(* CoDeSys 2.3.9.42 project: komp_new2.pro *)
(* Libraries: Standard.lib 2.12.10 17:48:34, SYSLIBCALLBACK.LIB 2.12.10 17:48:32 *)

(* PLC configuration (modules and I/O channels)
0750-1405 16 DI 24V DC 3.0ms [Type_1_16_Channels] node 0, in %IB24 out %QB0 {INTTypePAAssignment = PLC; INTTypeModule = plugged}
  S4_1 AT %IX12.0 [BOOLOnX_I] Ch_1 Digital input
  S4_2 AT %IX12.1 [BOOLOnX_I] Ch_2 Digital input
  S5_1 AT %IX12.2 [BOOLOnX_I] Ch_3 Digital input
  S5_2 AT %IX12.3 [BOOLOnX_I] Ch_4 Digital input
  S6_1 AT %IX12.4 [BOOLOnX_I] Ch_5 Digital input
  S6_2 AT %IX12.5 [BOOLOnX_I] Ch_6 Digital input
  S7_1 AT %IX12.6 [BOOLOnX_I] Ch_7 Digital input
  S7_2 AT %IX12.7 [BOOLOnX_I] Ch_8 Digital input
  S8_1 AT %IX12.8 [BOOLOnX_I] Ch_9 Digital input
  S8_2 AT %IX12.9 [BOOLOnX_I] Ch_10 Digital input
  S9_1 AT %IX12.10 [BOOLOnX_I] Ch_11 Digital input
  S9_2 AT %IX12.11 [BOOLOnX_I] Ch_12 Digital input
  S10_1 AT %IX12.12 [BOOLOnX_I] Ch_13 Digital input
  S10_2 AT %IX12.13 [BOOLOnX_I] Ch_14 Digital input
  S11_1 AT %IX12.14 [BOOLOnX_I] Ch_15 Digital input
  S11_2 AT %IX12.15 [BOOLOnX_I] Ch_16 Digital input
0750-1405 16 DI 24V DC 3.0ms [Type_1_16_Channels] node 1, in %IB24 out %QB0 {INTTypePAAssignment = PLC; INTTypeModule = plugged}
  S14_1 AT %IX13.0 [BOOLOnX_I] Ch_1 Digital input
  S14_2 AT %IX13.1 [BOOLOnX_I] Ch_2 Digital input
  S18_1 AT %IX13.2 [BOOLOnX_I] Ch_3 Digital input
  S18_2 AT %IX13.3 [BOOLOnX_I] Ch_4 Digital input
  S19_1 AT %IX13.4 [BOOLOnX_I] Ch_5 Digital input
  S19_2 AT %IX13.5 [BOOLOnX_I] Ch_6 Digital input
  _controlFazaDI AT %IX13.6 [BOOLOnX_I] Ch_7 Digital input
  _currentHighJD5DI AT %IX13.7 [BOOLOnX_I] Ch_8 Digital input
  _vacumContactOnDI AT %IX13.8 [BOOLOnX_I] Ch_9 Digital input
  _vacumContactOffDI AT %IX13.9 [BOOLOnX_I] Ch_10 Digital input
  __1pressLevelInDI AT %IX13.10 [BOOLOnX_I] Ch_11 Digital input
  __2pressLevelInDI AT %IX13.11 [BOOLOnX_I] Ch_12 Digital input
  __3pressLevelInDI AT %IX13.12 [BOOLOnX_I] Ch_13 Digital input
  __4pressLevelInDI AT %IX13.13 [BOOLOnX_I] Ch_14 Digital input
  _4pressLeveOutDI AT %IX13.14 [BOOLOnX_I] Ch_15 Digital input
  pressWaterDI AT %IX13.15 [BOOLOnX_I] Ch_16 Digital input
0750-1505 16 DO 24V DC 0.5A / LSS [Type_10_16_Channels] node 2, in %IB26 out %QB0 {INTTypePAAssignment = PLC; INTTypeModule = plugged}
  KM4_1 AT %QX0.0 [BOOLOnX_Q] Ch_1 Digital output
  KM4_2 AT %QX0.1 [BOOLOnX_Q] Ch_2 Digital output
  KM5_1 AT %QX0.2 [BOOLOnX_Q] Ch_3 Digital output
  KM5_2 AT %QX0.3 [BOOLOnX_Q] Ch_4 Digital output
  KM6_1 AT %QX0.4 [BOOLOnX_Q] Ch_5 Digital output
  KM6_2 AT %QX0.5 [BOOLOnX_Q] Ch_6 Digital output
  KM7_1 AT %QX0.6 [BOOLOnX_Q] Ch_7 Digital output
  KM7_2 AT %QX0.7 [BOOLOnX_Q] Ch_8 Digital output
  KM8_1 AT %QX0.8 [BOOLOnX_Q] Ch_9 Digital output
  KM8_2 AT %QX0.9 [BOOLOnX_Q] Ch_10 Digital output
  KM9_1 AT %QX0.10 [BOOLOnX_Q] Ch_11 Digital output
  KM9_2 AT %QX0.11 [BOOLOnX_Q] Ch_12 Digital output
  KM10_1 AT %QX0.12 [BOOLOnX_Q] Ch_13 Digital output
  KM10_2 AT %QX0.13 [BOOLOnX_Q] Ch_14 Digital output
  KM11_1 AT %QX0.14 [BOOLOnX_Q] Ch_15 Digital output
  KM11_2 AT %QX0.15 [BOOLOnX_Q] Ch_16 Digital output
0750-1505 16 DO 24V DC 0.5A / LSS [Type_10_16_Channels] node 3, in %IB28 out %QB0 {INTTypePAAssignment = PLC; INTTypeModule = plugged}
  KM14_1 AT %QX1.0 [BOOLOnX_Q] Ch_1 Digital output
  KM14_2 AT %QX1.1 [BOOLOnX_Q] Ch_2 Digital output
  KM18_1 AT %QX1.2 [BOOLOnX_Q] Ch_3 Digital output
  KM18_2 AT %QX1.3 [BOOLOnX_Q] Ch_4 Digital output
  readyWater AT %QX1.4 [BOOLOnX_Q] Ch_5 Digital output
  readyOil AT %QX1.5 [BOOLOnX_Q] Ch_6 Digital output
  _oilGate_1 AT %QX1.6 [BOOLOnX_Q] Ch_7 Digital output
  _oilGate_2 AT %QX1.7 [BOOLOnX_Q] Ch_8 Digital output
  KM2 AT %QX1.8 [BOOLOnX_Q] Ch_9 Digital output
  _rejimModeDO AT %QX1.9 [BOOLOnX_Q] Ch_10 Digital output
  KM1 AT %QX1.10 [BOOLOnX_Q] Ch_11 Digital output
  _PuskModeDO AT %QX1.11 [BOOLOnX_Q] Ch_12 Digital output
  _kompOnDO AT %QX1.12 [BOOLOnX_Q] Ch_13 Digital output
  _kompOffDO AT %QX1.13 [BOOLOnX_Q] Ch_14 Digital output
  _alarmLedDO_blink AT %QX1.14 [BOOLOnX_Q] Ch_15 Digital output
  _stopModeDO AT %QX1.15 [BOOLOnX_Q] Ch_16 Digital output
0753-0455 4 AI 4-20mA s.e. [Type_8_4_Channels] node 4, in %IB16 out %QB0 {INTTypePAAssignment = PLC; INTTypeModule = plugged}
  AT %IW0 [WORDOnW_I] Ch_1 Input word
  AT %IW1 [WORDOnW_I] Ch_2 Input word
  AT %IW2 [WORDOnW_I] Ch_3 Input word
  AT %IW3 [WORDOnW_I] Ch_4 Input word
0753-0455 4 AI 4-20mA s.e. [Type_8_4_Channels] node 5, in %IB16 out %QB0 {INTTypePAAssignment = PLC; INTTypeModule = plugged}
  AT %IW4 [WORDOnW_I] Ch_1 Input word
  AT %IW5 [WORDOnW_I] Ch_2 Input word
  AT %IW6 [WORDOnW_I] Ch_3 Input word
  AT %IW7 [WORDOnW_I] Ch_4 Input word
0753-0455 4 AI 4-20mA s.e. [Type_8_4_Channels] node 6, in %IB24 out %QB0 {INTTypePAAssignment = PLC; INTTypeModule = plugged}
  AT %IW8 [WORDOnW_I] Ch_1 Input word
  AT %IW9 [WORDOnW_I] Ch_2 Input word
  AT %IW10 [WORDOnW_I] Ch_3 Input word
  AT %IW11 [WORDOnW_I] Ch_4 Input word
0750-1405 16 DI 24V DC 3.0ms [Type_1_16_Channels] node 7, in %IB28 out %QB2 {INTTypePAAssignment = PLC; INTTypeModule = plugged}
  _konsovikMechanikMotor AT %IX14.0 [BOOLOnX_I] Ch_1 Digital input
  _emergencyStop AT %IX14.1 [BOOLOnX_I] Ch_2 Digital input
  _buttonStop AT %IX14.2 [BOOLOnX_I] Ch_3 Digital input
  _buttonRejim AT %IX14.3 [BOOLOnX_I] Ch_4 Digital input
  _buttonPusk AT %IX14.4 [BOOLOnX_I] Ch_5 Digital input
  _switchAuto AT %IX14.5 [BOOLOnX_I] Ch_6 Digital input
  _switchManual AT %IX14.6 [BOOLOnX_I] Ch_7 Digital input
  _emergencyStopMashZal AT %IX14.7 [BOOLOnX_I] Ch_8 Digital input
  gazaAnalizMashzal AT %IX14.8 [BOOLOnX_I] Ch_9 Digital input
  gazaAnaliz AT %IX14.9 [BOOLOnX_I] Ch_10 Digital input
  _pressOilMINDI AT %IX14.10 [BOOLOnX_I] Ch_11 Digital input
  _pressOilMAXDI AT %IX14.11 [BOOLOnX_I] Ch_12 Digital input
  pressOil_DI AT %IX14.12 [BOOLOnX_I] Ch_13 Digital input
  AT %IX14.13 [BOOLOnX_I] Ch_14 Digital input
  AT %IX14.14 [BOOLOnX_I] Ch_15 Digital input
  AT %IX14.15 [BOOLOnX_I] Ch_16 Digital input
Fieldbus variables [FB_VARS] node 1, in %IB0 out %QB0
Flag variables [FLAG_VARS] node 2, in %IB0 out %QB0
*)

(* Global variable list: _L *)
VAR_GLOBAL
	L11_PUSK : BOOL;
	L12_PUSK : BOOL;
	TO_LIST13: BOOL;

END_VAR

(* Global variable list: _S *)
VAR_GLOBAL
	_17S_1: BOOL;
	_16S_1: BOOL;
END_VAR

(* Global variable list: Global_Variables *)
VAR_GLOBAL
	_alarmLedDO : BOOL;
	alarm : ALARMS;
	_pressWaterDI : BOOL;
	_pressOil_DI : BOOL;
	_1pressLevelInDI : BOOL;
	_2pressLevelInDI : BOOL;
	_3pressLevelInDI : BOOL;
	_4pressLevelInDI : BOOL;
	(*waterPump1 : Pumps;
	waterPump2 : Pumps;
	oilPump1 : Pumps;
	oilPump2 : Pumps;
	_18gate : GateValve;
	_4gate : GateValve;
	_5gate : GateValve;
	_6gate : GateValve;
	_7gate : GateValve;
	_8gate : GateValve;
	_9gate : GateValve;
	_10gate : GateValve;
	_11gate : GateValve;
	_14gate : GateValve;
	_17gate : GateValve;
	_19gate : GateValve;
	_20gate : GateValve;
	heater : Heaters;
	komp : Compressor;

	wtrTimeWORD AT %QW256: WORD := 2;
	oilTimeWORD  AT %QW257: WORD := 2;

	MODE AT %QW280 : WORD;

	gate18TimeWORD  AT %IW258 :WORD := 2;
	gate4TimeWORD  AT %IW259 :WORD := 2;
	gate5TimeWORD  AT %IW260 :WORD := 2;
	gate6TimeWORD  AT %IW261 :WORD := 2;
	gate7TimeWORD  AT %IW262 :WORD := 2;
	gate8TimeWORD  AT %IW263 :WORD := 2;
	gate9TimeWORD  AT %IW264 :WORD := 2;
	gate10TimeWORD  AT %IW265 :WORD := 2;
	gate11TimeWORD  AT %IW266 :WORD := 2;
	gate14TimeWORD  AT %IW267 :WORD := 2;
	gate17TimeWORD  AT %QW268 :WORD := 2;
	gate17T3  AT %IW268 :WORD := 3;
	gate17T4  AT %MW268 :WORD := 4;
	
	wtrTime : TIME := T#2s;
	oilTime : TIME := T#2s;
	gate18Time  :TIME := T#2s;
	gate4Time  :TIME := T#2s;
	gate5Time  :TIME := T#2s;
	gate6Time  :TIME := T#2s;
	gate7Time  :TIME := T#2s;
	gate8Time  :TIME := T#2s;
	gate9Time  :TIME := T#2s;
	gate10Time :TIME := T#2s;
	gate11Time  :TIME := T#2s;
	gate14Time  :TIME := T#2s;
	gate17Time  :TIME := T#2s;

	goRejim AT %QX269.0 : BOOL;
	goPusk AT %QX269.1: BOOL;
	goSTOP AT %QX269.2 : BOOL;
	kompReady AT %QX269.3 : BOOL := FALSE;
	isOK AT %QX269.4: BOOL := TRUE;

	_4gate_open  AT %IX269.5 : BOOL;
	_4gate_close  AT %IX269.6 : BOOL;
	_5gate_open  AT %IX269.7 : BOOL;
	_5gate_close  AT %IX269.8 : BOOL;
	_6gate_open  AT %IX269.9 : BOOL;
	_6gate_close  AT %IX269.10 : BOOL;
	_7gate_open  AT %IX269.11 : BOOL;
	_7gate_close  AT %IX269.12 : BOOL;
	_8gate_open  AT %IX269.13 : BOOL;
	_8gate_close  AT %IX269.14 : BOOL;
	_9gate_open  AT %IX269.15 : BOOL;
	_9gate_close  AT %IX270.0 : BOOL;
	_10gate_open  AT %IX270.1 : BOOL;
	_10gate_close  AT %IX270.2 : BOOL;
	_11gate_open  AT %IX270.3 : BOOL;
	_11gate_close  AT %IX270.4 : BOOL;
	_14gate_open  AT %IX270.5 : BOOL;
	_14gate_close  AT %IX270.6 : BOOL;
	_18gate_open  AT %IX270.7 : BOOL;
	_18gate_close  AT %IX270.8 : BOOL;
	_19gate_open  AT %IX270.9 : BOOL;
	_19gate_close  AT %IX270.10 : BOOL;
	_20gate_open  AT %IX270.11 : BOOL;
	_20gate_close  AT %IX270.12 : BOOL;
	oilPump1_run  AT %IX270.13 : BOOL;
	oilPump2_run  AT %IX270.14 : BOOL;
	waterPump1_run  AT %IX270.15 : BOOL;
	waterPump2_run  AT %IX271.0 : BOOL;
	komp_run  AT %IX271.1 : BOOL;
	komp_stop  AT %IX271.2 : BOOL;
	autoManual  AT %IX272.0 : BOOL;
	*)


END_VAR

(* Global variable list: K *)
VAR_GLOBAL

	K01: BOOL;
	K1: BOOL;
	K2: BOOL;
	K3: BOOL;
	K4: BOOL;
	K5: BOOL;
	K6 : BOOL;
	K7 : BOOL;
	K8 : BOOL;
	K13 : BOOL;
	K14: BOOL;
	K15: BOOL;
END_VAR

(* Global variable list: KM *)
VAR_GLOBAL

	TRM7: BOOL := TRUE;
	KM3: BOOL; (*Nagrev gaza*)
(*
	KM1: BOOL; (* suv nasos*)
	KM2: BOOL; (*maslo nasos*)
	
	KM4_1: BOOL;  (*Zadvijka 4 katushka ochish*)
	KM4_2: BOOL;  (*Zadvijka 4 katushka YOPISH*)
	KM5_1: BOOL;  (*Zadvijka 5 katushka ochish*)
	KM5_2: BOOL;  (*Zadvijka 5 katushka ochish*)
	KM6_1 : BOOL; (*Zadvijka 6 katushka ochish*)
	KM6_2 : BOOL; (*Zadvijka 6 katushka YOPISH*)
	KM7_1: BOOL; (*Zadvijka 7 katushka ochish*)
	KM7_2: BOOL;  (*Zadvijka 7 katushka YOPISH*)
	KM8_1: BOOL; (*Zadvijka 8 katushka ochish*)
	KM8_2: BOOL; (*Zadvijka 8 katushka YOPISH*)
	KM9_1: BOOL;  (*Zadvijka 9 katushka ochish*)
	KM9_2: BOOL;  (*Zadvijka 9 katushka YOPISH*)
	KM10_1: BOOL;  (*Zadvijka 10 katushka ochish*)
	KM10_2: BOOL; (*Zadvijka 10 katushka YOPISH*)
	KM11_1: BOOL; (*Zadvijka 11 katushka ochish*)
	KM11_2: BOOL; (*Zadvijka 11 katushka YOPISH*)
	KM13_1: BOOL;  (*Zadvijka 13 katushka ochish*)
	KM13_2: BOOL; (*Zadvijka 13 katushka YOPISH*)
	KM14_1: BOOL;  (*Zadvijka 14 katushka ochish*)
	KM14_2: BOOL;  (*Zadvijka 14 katushka YOPISH*)
	KM15_1 : BOOL;  (*Zadvijka 15 katushka ochish*)
	KM15_2 : BOOL; (*Zadvijka 15 katushka YOPISH*)
	
	KM18_1 : BOOL; (*Zadvijka 18 katushka ochish*)
	KM18_2 : BOOL;	(*Zadvijka 18 katushka YOPISH*)
*)
	KM16_1: BOOL;  (*Zadvijka 16 katushka ochish*)
	KM16_2: BOOL; (*Zadvijka 16 katushka YOPISH*)
	KM17_1: BOOL; (*Zadvijka 17 katushka ochish*)
	KM17_2: BOOL; (*Zadvijka 17 katushka YOPISH*)
END_VAR

(* Global variable list: P *)
VAR_GLOBAL

	P0: BOOL;

	P1 : BOOL; 	(*GOTOVNOST*)
	P2 : BOOL; 	(*REJIM*)
	P3: BOOL; 	(* STOP kompressor*)
	P4 : BOOL;
	P5 : BOOL;
	P6 : BOOL;	 (* EKM vodinoy nasos*)
	P7 : BOOL; 	(* EKM maslo nasos*)


END_VAR

(* Global variable list: RV *)
VAR_GLOBAL


	RV3: BOOL;
	RV4: BOOL;
	RV5: BOOL;
	RV13: BOOL;
	RV15: BOOL;

	RV3TON: TON;
	RV4TON: TON;
	RV5TON: TON;
	RV13TON : TON;
	RV15TON : TON;


END_VAR

(* Global variable list: V_MODBUS *)
VAR_GLOBAL

	S4_1MB AT %MX100.0 : BOOL;
	S4_2MB AT %MX100.1 : BOOL;
	S5_1MB AT %MX100.2 : BOOL;
	S5_2MB AT %MX100.3 : BOOL;
	S6_1MB AT %MX100.4 : BOOL;
	S6_2MB AT %MX100.5 : BOOL;
	S7_1MB AT %MX100.6 : BOOL;
	S7_2MB AT %MX100.7 : BOOL;
	S8_1MB AT %MX100.8 : BOOL;
	S8_2MB AT %MX100.9 : BOOL;
	S9_1MB AT %MX100.10 : BOOL;
	S9_2MB AT %MX100.11 : BOOL;
	S10_1MB AT %MX100.12 : BOOL;
	S10_2MB AT %MX100.13 : BOOL;
	S11_1MB AT %MX100.14 : BOOL;
	S11_2MB AT %MX100.15 : BOOL;
	S14_1MB AT %MX101.0 : BOOL;
	S14_2MB AT %MX101.1 : BOOL;
	S18_1MB AT %MX101.2 : BOOL;
	S18_2MB AT %MX101.3 : BOOL;
	S19_1MB AT %MX101.4 : BOOL;
	S19_2MB AT %MX101.5 : BOOL;
	controlFazaDIMB AT %MX101.6 : BOOL;
	currentHighJD5DIMB AT %MX101.7 : BOOL;
	vacumContactOnDIMB AT %MX101.8 : BOOL;
	vacumContactOffDIMB AT %MX101.9 : BOOL;
	press1LevelInDIMB AT %MX101.10 : BOOL;
	press2LevelInDIMB AT %MX101.11 : BOOL;
	press3LevelInDIMB AT  %MX101.12 : BOOL;
	press4LevelInDIMB AT %MX101.13 : BOOL;
	press4LevelOutDIMB AT %MX101.14 : BOOL;
	pressWaterDIMB AT  %MX101.15 : BOOL;
	KM4_1MB AT %MX102.0 : BOOL;
	KM4_2MB AT %MX102.1 : BOOL;
	KM5_1MB AT %MX102.2 : BOOL;
	KM5_2MB AT %MX102.3 : BOOL;
	KM6_1MB AT %MX102.4 : BOOL;
	KM6_2MB AT %MX102.5 : BOOL;
	KM7_1MB AT %MX102.6 : BOOL;
	KM7_2MB AT %MX102.7 : BOOL;
	KM8_1MB AT %MX102.8 : BOOL;
	KM8_2MB AT %MX102.9 : BOOL;
	KM9_1MB AT %MX102.10 : BOOL;
	KM9_2MB AT %MX102.11 : BOOL;
	KM10_1MB AT %MX102.12 : BOOL;
	KM10_2MB AT %MX102.13 : BOOL;
	KM11_1MB AT %MX102.14 : BOOL;
	KM11_2MB AT %MX102.15 : BOOL;

	KM14_1MB AT %MX103.0 : BOOL;
	KM14_2MB AT %MX103.1 : BOOL;
	KM18_1MB AT %MX103.2 : BOOL;
	KM18_2MB AT %MX103.3 : BOOL;
	KM19_1MB AT %MX103.4 : BOOL;
	KM19_2MB AT %MX103.5 : BOOL;
	KM1_MB AT %MX103.6 : BOOL;
	KM2_MB AT %MX103.7 : BOOL;
	kompOnDO_MB AT %MX103.8 : BOOL;
	kompOffDO_MB AT %MX103.9 : BOOL;
	alarmLedDO_MB AT %MX103.10 : BOOL;
	stopModeDO_MB AT %MX103.11 : BOOL;
	acknowledgment_MB AT %MX103.12 : BOOL;
	gazaAnaliz_MB AT %MX103.12 : BOOL;
	gazaAnalizMashzal_MB  AT %MX103.13 : BOOL;
	serviceMODE_MB AT %MX103.14 : BOOL;
	SB3 AT %MX104.0: BOOL;  (*PUSK VODA knopka*)
	SB4 AT %MX104.1: BOOL;  (*STOP VODA knopka*)
	SB5 AT %MX104.2: BOOL; (*PUSK MASLO knopka*)
	SB6 AT %MX104.3: BOOL; (*STOP MASLO knopka*)
	SB7 AT %MX104.4: BOOL; (*PUSK NAGREV knopka*)
	SB8 AT %MX104.5: BOOL; (*STOP NAGREV knopka*)
	SB9 AT %MX104.6: BOOL; (*Zadvijka 4 ochish knopka*)
	SB10 AT %MX104.7: BOOL;  (*Zadvijka  4  YOPISH   knopka*)
	SB11 AT %MX104.8: BOOL; (*Zadvijka 5 ochish knopka*)
	SB12 AT %MX104.9: BOOL; (*Zadvijka 5 YOPISH knopka*)
	SB13 AT %MX104.10: BOOL; (*Zadvijka 6 ochish knopka*)
	SB14 AT %MX104.11: BOOL;  (*Zadvijka 6 YOPISH knopka*)
	SB15 AT %MX104.12: BOOL;  (*Zadvijka 7 ochish knopka*)
	SB16 AT %MX104.13: BOOL; (*Zadvijka 7 YOPISH knopka*)
	SB17 AT %MX104.14: BOOL;  (*Zadvijka 8 ochish knopka*)
	SB18 AT %MX104.15: BOOL; (*Zadvijka 8 YOPISH knopka*)

	SB19 AT %MX105.0: BOOL;	 (*Zadvijka 9 ochish knopka*)
	SB20 AT %MX105.1: BOOL;  (*Zadvijka 9 YOPISH knopka*)
	SB21 AT %MX105.2: BOOL;	 (*Zadvijka 10 ochish knopka*)
	SB22 AT %MX105.3: BOOL; (*Zadvijka 10 YOPISH knopka*)
	SB23 AT %MX105.4: BOOL; (*Zadvijka 11 ochish knopka*)
	SB24 AT %MX105.5: BOOL; (*Zadvijka 11 YOPISH knopka*)
	SB25 AT %MX105.6: BOOL;  (*Zadvijka 14 ochish knopka*)
	SB26 AT %MX105.7: BOOL;  (*Zadvijka 14 YOPISH knopka*)
	SB29 AT %MX105.8: BOOL;  (*Zadvijka 18 ochish knopka*)
	SB30 AT %MX105.9: BOOL;   (*Zadvijka 18 YOPISH knopka*)
	SB32 AT %MX105.10: BOOL; (*Zadvijka 16 YOPISH knopka*)
	SBA41 AT %IX14.12: BOOL; (* Avariyniy stop*)
	SBA41_MB AT %MX105.11: BOOL; (* Avariyniy stop*)
	SB42 AT  %IX14.3: BOOL;	 (* knopka REJIM*)
	SB42_MB AT  %MX105.12: BOOL;	 (* knopka REJIM*)
	SB43 AT %IX14.4: BOOL; (* knopka PUSK*)
	SB43_MB AT %MX105.13: BOOL; (* knopka PUSK*)
	SB44 AT %IX14.2: BOOL; (*Kompressor STOP*)
	SB44_MB AT %MX105.14: BOOL; (*Kompressor STOP*)
	(*SB53_1 : BOOL := TRUE; (*obshiy stop zadvijek *)*)
	SB53_1 AT %IX14.2: BOOL; (*obshiy stop zadvijek *)
	SB53_1MB AT %MX105.15 : BOOL; (*obshiy stop zadvijek *)

	(*SBZ AT %IX15.1: BOOL; (*AVARIYNIY STOP MASH ZALA*)*)
	SBZ_MB AT %MX106.0: BOOL; (*AVARIYNIY STOP MASH ZALA*)
	SA45_1MB AT %MX106.1: BOOL;
	SA45_2MB AT %MX106.2: BOOL;
	SB28 : BOOL;  (*Zadvijka 17 YOPISH knopka*)
	SA45_1 : BOOL; (*Auto mode switch*)
	(*SA45_1 AT %IX14.5: BOOL; (*Auto mode switch*)*)
	(*SA45_2 AT %IX14.1: BOOL; (*Emergency stop*)*)
	SA45_2 : BOOL; (*Emergency stop*)



	pressOilMINDI_MB AT %MX107.0 : BOOL;
	rejimModeDO_MB AT  %MX107.1 : BOOL;
	pressOilMAXDI_MB AT %MX107.2 : BOOL;
	puskModeDO_MB AT %MX107.3 :BOOL;
	pressOilDI_MB AT %MX107.4 : BOOL;

	konsovikMechanikMotor AT %MX108.0 : BOOL;
	emergencyStop_MB AT %MX108.1 : BOOL;
	buttonStop_MB AT %MX108.2 : BOOL;
	buttonRejim_MB AT %MX108.3 : BOOL;
	buttonPusk_MB AT %MX108.4 : BOOL;
	switchAuto_MB AT %MX108.5 : BOOL;
	switchManual_MB AT %MX108.6 : BOOL;
	emergencyStopmashZal_MB AT %MX108.7 : BOOL;
	alarrm4levelTemp_MB AT %MX108.8 : BOOL;


	analog1 AT %MW120 : REAL;
	analog2 AT %MW122 : REAL;
	analog3 AT %MW124 : REAL;
	analog4 AT %MW126 : REAL;
	analog5 AT %MW128 : REAL;
	analog6 AT %MW130 : REAL;
	analog7 AT %MW132 : REAL;
	analog8 AT %MW134 : REAL;
	analog9 AT %MW136 : REAL;
	analog10 AT %MW138 : REAL;
	analog11 AT %MW140 : REAL;
	analog12 AT %MW142 : REAL;



END_VAR
VAR_GLOBAL RETAIN PERSISTENT
	analog1SP AT %MW144 : REAL := 250; (*reg 12433*)
	analog2SP AT %MW146 : REAL := 10; (*reg 12435*)
	analog3SP AT %MW148 : REAL := 0.8; (*reg 12437*)
	analog4SP AT %MW150 : REAL := 3.5; (*reg 12439*)

	analog5SP AT %MW152 : REAL := 22; (*reg 12441*)
	analog6SP AT %MW154 : REAL := 64; (*reg 12443*)
	analog7SP AT %MW156 : REAL := 178; (*reg 12445*)
	analog8SP AT %MW158 : REAL := 275; (*reg 12447*)

	analog9SP AT %MW160 : REAL := 1.5; (*reg 12449*)
	analog10SP AT %MW162 : REAL := 150; (*reg 12449*)



END_VAR

(* Data type *)
		TYPE ALARMS :
STRUCT
	gate18NotOpen AT %MX109.0 : BOOL; (* reg 12398.00*)
	gate18NotClose AT %MX109.1 : BOOL; (* reg 12398.01*)

	gate4NotOpen AT %MX109.2 : BOOL; (* reg 12398.02*)
	gate4NotClose AT %MX109.3 : BOOL; (* reg 12398.03*)

	gate5NotOpen AT %MX109.4 : BOOL; (* reg 12398.04*)
	gate5NotClose AT %MX109.5 : BOOL; (* reg 12398.05*)

	gate6NotOpen AT %MX109.6 : BOOL; (* reg 12398.06*)
	gate6NotClose AT %MX109.7 : BOOL; (* reg 12398.07*)

	gate7NotOpen AT %MX109.8 : BOOL; (* reg 12398.08*)
	gate7NotClose AT %MX109.9 : BOOL; (* reg 12398.09*)

	gate8NotOpen AT %MX109.10 : BOOL; (* reg 12398.10*)
	gate8NotClose AT %MX109.11 : BOOL; (* reg 12398.11*)

	gate9NotOpen  AT %MX109.12: BOOL; (* reg 12398.12*)
	gate9NotClose AT %MX109.13 : BOOL; (* reg 12398.13*)

	gate10NotOpen AT %MX109.14 : BOOL; (* reg 12398.14*)
	gate10NotClose AT %MX109.15 : BOOL; (* reg 12398.15*)

	gate11NotOpen AT %MX110.0 : BOOL; (* reg 12399.00*)
	gate11NotClose  AT %MX110.1: BOOL; (* reg 12399.01*)

	gate14NotOpen AT %MX110.2 : BOOL; (* reg 12399.02*)
	gate14NotClose AT %MX110.3 : BOOL; (* reg 12399.03*)
	alarmGazAnaliz AT  %MX110.4 : BOOL; (* reg 12399.04*)
END_STRUCT
END_TYPE

(* POU PLC_PRG, ST *)
PROGRAM PLC_PRG
VAR
END_VAR
SA45_1 := _switchAuto;
SA45_2 := _emergencyStop AND _emergencyStopMashZal ;
translate();
IF (_switchAuto) THEN
	L05();
	L08();
	L09();
	L10();
	L11();
	L12();
	L13();
	L14();
	L15();
	L16();
END_IF;
gatesAlarm();
start_or_stop();
E_STOP();
blink();
END_PROGRAM

(* POU translate, ST *)
PROGRAM translate
VAR

	K3: BOOL;
	vaqt : TIME := T#2s;
	SC1: SCALE;
	SC2: SCALE;
	SC3: SCALE;
	SC4: SCALE;
	SC5: SCALE;
	SC6: SCALE;
	SC7: SCALE;
	SC8: SCALE;
	SC9: SCALE;
	SC10: SCALE;
	tmrWater : TOF;
	tmrOil: TOF;
	SC11: SCALE;
	SC12: SCALE;
	trig: R_TRIG;
	tonn : ARRAY [1..5] OF TON;
	vaqtt : TIME := T#500ms;
END_VAR
VAR (* helpers for the ST form of the networks *)
	_p1 : BOOL;
END_VAR
MODBUS();
gazaAnaliz_MB := gazaAnaliz;
ANALOG();
ERRORS();
IF (analog1 > analog1SP) THEN
	TRM7 := TRUE;
END_IF;
IF (analog1 < analog1SP - 5) THEN
	TRM7 := FALSE;
END_IF;

K01 := analog3 < analog2SP;
K1 := _1pressLevelInDI;
K2 := _2pressLevelInDI;
K3 := _3pressLevelInDI;
K4 := _4pressLevelInDI;
 _rejimModeDO := (P1 AND _vacumContactOffDI) OR P2;
_stopModeDO := NOT  P1 AND  _vacumContactOffDI;
_PuskModeDO := _vacumContactOnDI;
(*
IF (kompOnDO_MB = TRUE) THEN
	_kompOnDO :=  kompOnDO_MB;
ELSE
	_kompOnDO := FALSE;
END_IF;
IF (kompOffDO_MB = TRUE ) THEN
	_kompOffDO :=  kompOffDO_MB;
ELSE
	_kompOffDO := FALSE;
END_IF
*)
END_PROGRAM
ACTION ANALOG:
		SC1(IN := %IW0, MIN_VALUE := 0, MAX_VALUE := 400, OUT => analog1); (*Akummulator pressure*)
		SC2(IN := %IW1, MIN_VALUE := 0, MAX_VALUE := 400, OUT => analog2); (*Gas pressure 1 level*)
		SC3(IN := %IW2, MIN_VALUE := 0, MAX_VALUE := 400, OUT => analog3);  (*Incomming gas pressure*)
		SC4(IN := %IW3, MIN_VALUE := 0, MAX_VALUE := 400, OUT => analog4);  (*Pressure 2 level*)

		SC5(IN := %IW4,MIN_VALUE := 0, MAX_VALUE := 400,  OUT => analog5); (*Pressure 3 level*)
		SC6(IN := %IW5,MIN_VALUE := 0, MAX_VALUE := 250,  OUT => analog6);     (*Pressure water*)
		SC7(IN := %IW6, MIN_VALUE := 0, MAX_VALUE := 400, OUT => analog7); (*Pressure 4 level*)
		SC8(IN := %IW7, MIN_VALUE := 0, MAX_VALUE := 250, OUT => analog8);   (*Pressure after filtr*)

		SC9(IN := %IW8, MIN_VALUE := 0, MAX_VALUE := 16, OUT => analog9);    (*Pressure before filtr*)
		SC10(IN := %IW9, MIN_VALUE := -50, MAX_VALUE := 150, OUT => analog10); (*Temperture 4 level*)
		SC11(IN := %IW10, MIN_VALUE := -50, MAX_VALUE := 150, OUT => analog11); (*Temperture oil*)
		SC12(IN := %IW11, MIN_VALUE := 0, MAX_VALUE := 1000, OUT => analog12);  (*Motor currency*)
		tmrWater(IN := analog6  > analog3SP, PT := T#5s );
		_pressWaterDI :=  tmrWater.Q;
		readyWater := _pressWaterDI;
		tmrOil(IN := (analog9 > analog4SP AND  analog8 > analog9SP ), PT := T#5s);
		_pressOil_DI    :=  tmrOil.Q;
 		readyOil := _pressOil_DI;
		tonn[1](IN := analog2 >  analog5SP, PT := vaqtt);
		tonn[2](IN := analog4 >  analog6SP, PT := vaqtt);
		tonn[3](IN := analog5 >  analog7SP, PT := vaqtt);
		tonn[4](IN := analog7 >  analog8SP, PT := vaqtt);
		tonn[5](IN := analog10 >  analog10SP, PT := vaqtt);
		_1pressLevelInDI   := tonn[1].Q  ;
		_2pressLevelInDI   := tonn[2].Q;
		_3pressLevelInDI   := tonn[3].Q;
		_4pressLevelInDI   := tonn[4].Q;
		alarrm4levelTemp_MB    := tonn[5].Q;;
END_ACTION
ACTION ERRORS:
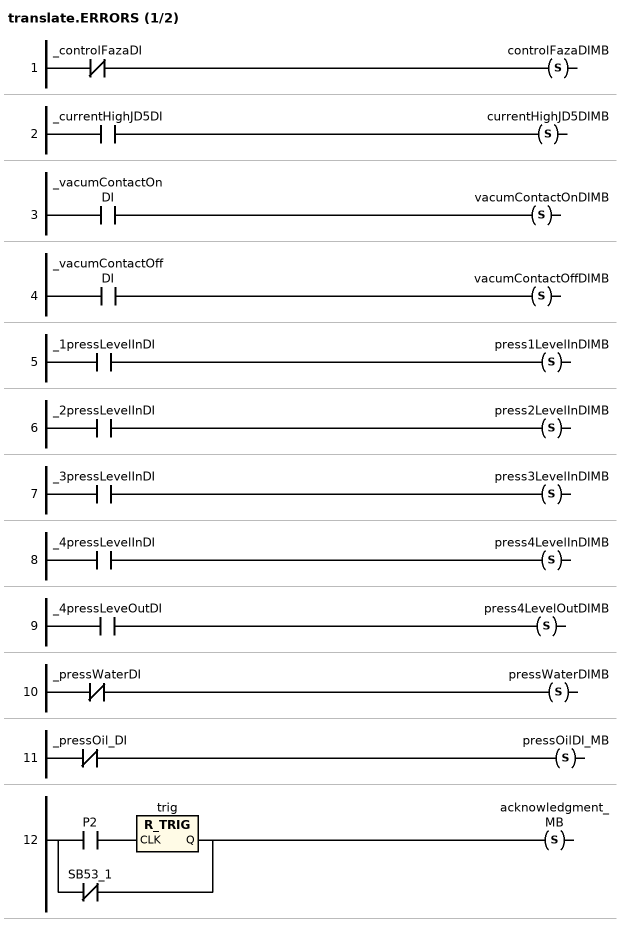
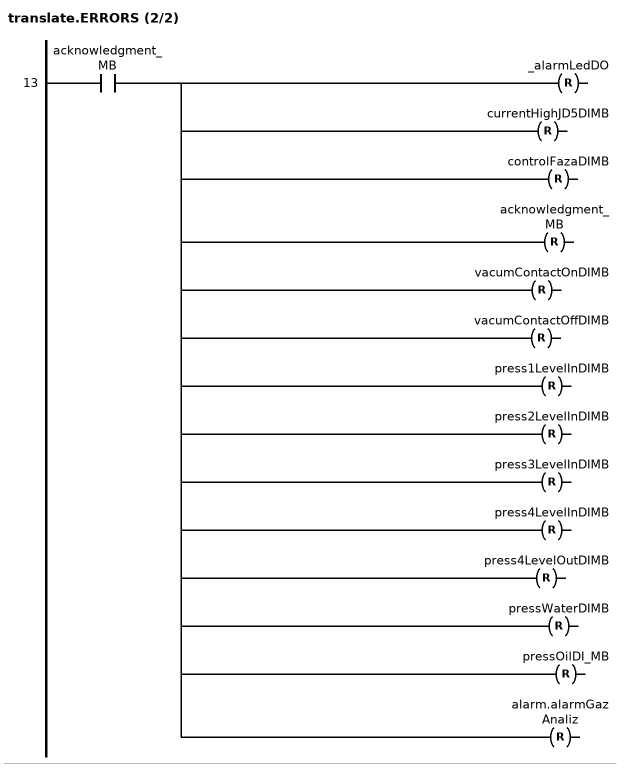
_LD_ (* Ladder Diagram *)
NETWORK 1
	[/_controlFazaDI] --- (S controlFazaDIMB)
NETWORK 2
	[_currentHighJD5DI] --- (S currentHighJD5DIMB)
NETWORK 3
	[_vacumContactOnDI] --- (S vacumContactOnDIMB)
NETWORK 4
	[_vacumContactOffDI] --- (S vacumContactOffDIMB)
NETWORK 5
	[_1pressLevelInDI] --- (S press1LevelInDIMB)
NETWORK 6
	[_2pressLevelInDI] --- (S press2LevelInDIMB)
NETWORK 7
	[_3pressLevelInDI] --- (S press3LevelInDIMB)
NETWORK 8
	[_4pressLevelInDI] --- (S press4LevelInDIMB)
NETWORK 9
	[_4pressLeveOutDI] --- (S press4LevelOutDIMB)
NETWORK 10
	[/_pressWaterDI] --- (S pressWaterDIMB)
NETWORK 11
	[/_pressOil_DI] --- (S pressOilDI_MB)
NETWORK 12
	{ [P2] - trig:R_TRIG(CLK: *) | [/SB53_1] } --- (S acknowledgment_MB)
NETWORK 13
	[acknowledgment_MB] --- (R _alarmLedDO) (R currentHighJD5DIMB) (R controlFazaDIMB) (R acknowledgment_MB) (R vacumContactOnDIMB) (R vacumContactOffDIMB) (R press1LevelInDIMB) (R press2LevelInDIMB) (R press3LevelInDIMB) (R press4LevelInDIMB) (R press4LevelOutDIMB) (R pressWaterDIMB) (R pressOilDI_MB) (R alarm.alarmGazAnaliz)
_END_LD_
(* the same logic as Structured Text *)
(* Network 1 *)
IF NOT _controlFazaDI THEN controlFazaDIMB := TRUE; END_IF;
(* Network 2 *)
IF _currentHighJD5DI THEN currentHighJD5DIMB := TRUE; END_IF;
(* Network 3 *)
IF _vacumContactOnDI THEN vacumContactOnDIMB := TRUE; END_IF;
(* Network 4 *)
IF _vacumContactOffDI THEN vacumContactOffDIMB := TRUE; END_IF;
(* Network 5 *)
IF _1pressLevelInDI THEN press1LevelInDIMB := TRUE; END_IF;
(* Network 6 *)
IF _2pressLevelInDI THEN press2LevelInDIMB := TRUE; END_IF;
(* Network 7 *)
IF _3pressLevelInDI THEN press3LevelInDIMB := TRUE; END_IF;
(* Network 8 *)
IF _4pressLevelInDI THEN press4LevelInDIMB := TRUE; END_IF;
(* Network 9 *)
IF _4pressLeveOutDI THEN press4LevelOutDIMB := TRUE; END_IF;
(* Network 10 *)
IF NOT _pressWaterDI THEN pressWaterDIMB := TRUE; END_IF;
(* Network 11 *)
IF NOT _pressOil_DI THEN pressOilDI_MB := TRUE; END_IF;
(* Network 12 *)
trig(CLK := P2);
IF trig.Q OR NOT SB53_1 THEN acknowledgment_MB := TRUE; END_IF;
(* Network 13 *)
_p1 := acknowledgment_MB;
IF _p1 THEN _alarmLedDO := FALSE; currentHighJD5DIMB := FALSE; controlFazaDIMB := FALSE; acknowledgment_MB := FALSE; vacumContactOnDIMB := FALSE; vacumContactOffDIMB := FALSE; press1LevelInDIMB := FALSE; press2LevelInDIMB := FALSE; press3LevelInDIMB := FALSE; press4LevelInDIMB := FALSE; press4LevelOutDIMB := FALSE; pressWaterDIMB := FALSE; pressOilDI_MB := FALSE; alarm.alarmGazAnaliz := FALSE; END_IF;
END_ACTION
ACTION MODBUS:
S4_1MB := S4_1;
S4_2MB := S4_2;
S5_1MB := S5_1;
S5_2MB := S5_2;
S6_1MB := S6_1;
S6_2MB := S6_2;
S7_1MB := S7_1;
S7_2MB := S7_2;
S8_1MB := S8_1;
S8_2MB := S8_2;
S9_1MB := S9_1;
S9_2MB := S9_2;
S10_1MB := S10_1;
S10_2MB := S10_2;
S11_1MB := S11_1;
S11_2MB := S11_2;
S14_1MB := S14_1;
S14_2MB := S14_2;
S18_1MB := S18_1;
S18_2MB := S18_2;
S19_1MB := S19_1;
S19_2MB := S19_2;


KM4_1MB := KM4_1;
KM4_2MB := KM4_2;
KM5_1MB := KM5_1;
KM5_2MB := KM5_2;
KM6_1MB := KM6_1;
KM6_2MB := KM6_2;
KM7_1MB := KM7_1;
KM7_2MB := KM7_2;
KM8_1MB := KM8_1;
KM8_2MB := KM8_2;
KM9_1MB := KM9_1;
KM9_2MB := KM9_2;
KM10_1MB := KM10_1;
KM10_2MB := KM10_2;
KM11_1MB := KM11_1;
KM11_2MB := KM11_2;

KM14_1MB := KM14_1;
KM14_2MB := KM14_2;
KM18_1MB := KM18_1;
KM18_2MB := KM18_2;
KM19_1MB := _oilGate_1;
KM19_2MB := _oilGate_2;
KM1_MB := KM1;
KM2_MB := KM2;
(*
kompOnDO_MB := _kompOnDO;
kompOffDO_MB := _kompOffDO;*)
alarmLedDO_MB := _alarmLedDO;
stopModeDO_MB := _stopModeDO;

konsovikMechanikMotor := _konsovikMechanikMotor;
emergencyStop_MB := NOT _emergencyStop;
SBA41_MB := SBA41;
SB42_MB := SB42;
SB43_MB := SB43;
SB44_MB := SB44;
SB53_1MB := SB53_1;




buttonStop_MB := _buttonStop;
buttonRejim_MB := _buttonRejim;
buttonPusk_MB := _buttonPusk;
switchAuto_MB := _switchAuto;
switchManual_MB := _switchManual;
emergencyStopmashZal_MB := NOT  _emergencyStopMashZal;
END_ACTION

(* POU SCALE, ST *)
FUNCTION_BLOCK SCALE
VAR_INPUT
	IN : WORD;
	MIN_VALUE : REAL := 4;
	MAX_VALUE : REAL := 20;
END_VAR
VAR_OUTPUT
	OUT : REAL;
END_VAR
VAR
	T : REAL;
	t2 : REAL;
	n : INT := 0;
	tp1 : TP;
	reset :BOOL;
	vaqt : TIME  := T#300ms;
END_VAR
T := WORD_TO_REAL(IN);
tp1(in := reset, PT := vaqt);
IF (tp1.Q) THEN
	n := n + 1;
	T2 := T2 +  (MAX_VALUE - MIN_VALUE) * T / 32767 +  MIN_VALUE;
ELSE
	out := T2 / n;
	n := 0;
	T2 := 0;
END_IF;
reset := NOT tp1.Q;
END_FUNCTION_BLOCK

(* POU alarm, CFC *)
FUNCTION_BLOCK alarm
VAR_INPUT
	start : BOOL;
	vaqtSekund : WORD := 45;
	konsevik : BOOL;
END_VAR
VAR_OUTPUT
	out : BOOL;
END_VAR
VAR
	TP: TON;
	temp: BOOL;
	rtrig: R_TRIG;
END_VAR
VAR (* helpers for the ST form of the networks *)
	_t8 : BOOL;
	_t4 : TIME;
END_VAR
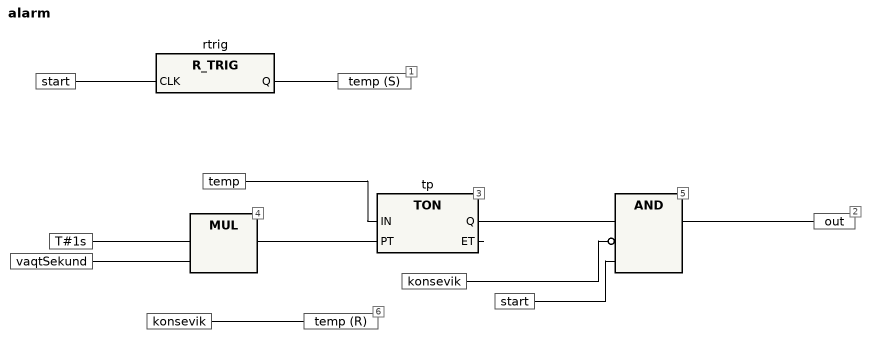
_CFC_ (* Continuous Function Chart, elements in execution order *)
#0 rtrig:R_TRIG(CLK: start)
#1 S temp <= #0.Q
#2 out <= #5
#3 tp:TON(IN: temp, PT: #4)
#4 MUL(T#1s, vaqtSekund)
#5 AND(#3.Q, NOT konsevik, start)
#6 R temp <= konsevik
_END_CFC_
(* the same logic as Structured Text *)
rtrig(CLK := start);
IF rtrig.Q THEN temp := TRUE; END_IF;
out := _t8;
tp(IN := temp, PT := _t4);
_t4 := T#1s * vaqtSekund;
_t8 := tp.Q AND NOT konsevik AND start;
IF konsevik THEN temp := FALSE; END_IF;
END_FUNCTION_BLOCK

(* POU L05, CFC *)
PROGRAM L05
VAR
	_kompOffDO000000000: BOOL;
	t6AfterTON : TON;

END_VAR
VAR (* helpers for the ST form of the networks *)
	_t5 : BOOL;
	_t6 : BOOL;
	_t36 : BOOL;
	_t141 : BOOL;
	_t46 : BOOL;
END_VAR
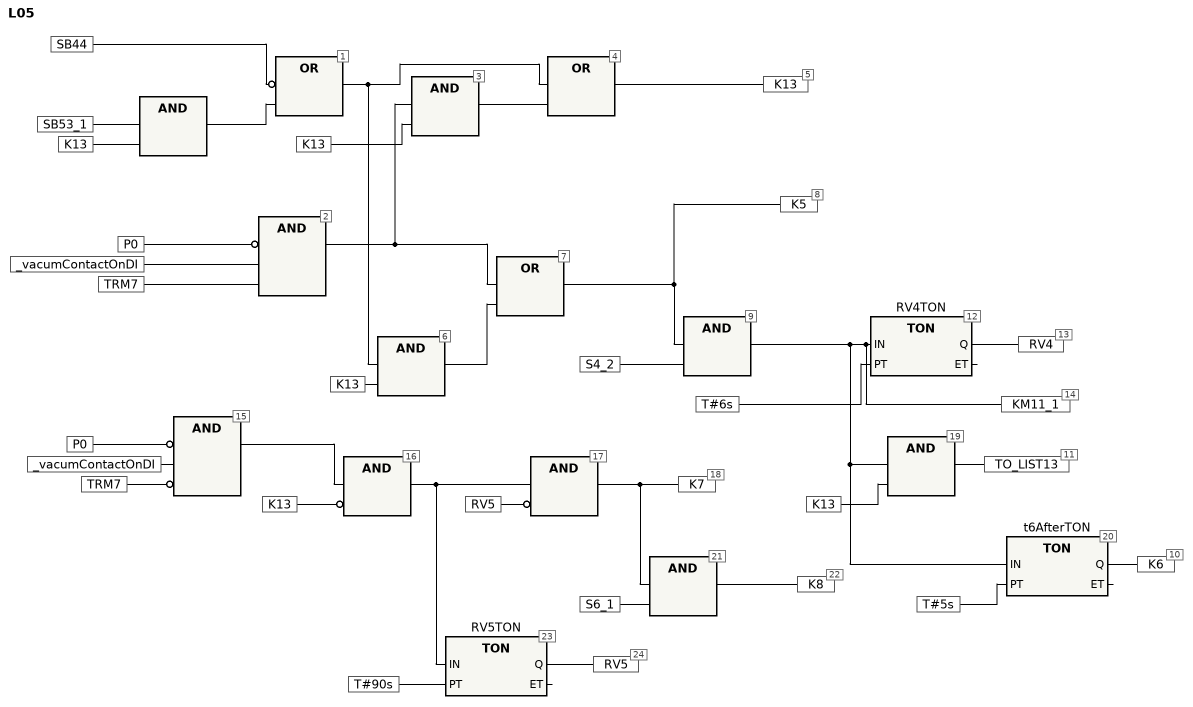
_CFC_ (* Continuous Function Chart, elements in execution order *)
#0 AND(SB53_1, K13)
#1 OR(NOT SB44, #0)
#2 AND(NOT P0, _vacumContactOnDI, TRM7)
#3 AND(#2, K13)
#4 OR(#1, #3)
#5 K13 <= #4
#6 AND(#1, K13)
#7 OR(#2, #6)
#8 K5 <= #7
#9 AND(#7, S4_2)
#10 K6 <= #20.Q
#11 TO_LIST13 <= #19
#12 RV4TON:TON(IN: #9, PT: T#6s)
#13 RV4 <= #12.Q
#14 KM11_1 <= #9
#15 AND(NOT P0, _vacumContactOnDI, NOT TRM7)
#16 AND(#15, NOT K13)
#17 AND(#16, NOT RV5)
#18 K7 <= #17
#19 AND(#9, K13)
#20 t6AfterTON:TON(IN: #9, PT: T#5s)
#21 AND(#17, S6_1)
#22 K8 <= #21
#23 RV5TON:TON(IN: #16, PT: T#90s)
#24 RV5 <= #23.Q
_END_CFC_
(* the same logic as Structured Text *)
_t5 := NOT SB44 OR (SB53_1 AND K13);
_t6 := NOT P0 AND _vacumContactOnDI AND TRM7;
K13 := _t5 OR (_t6 AND K13);
K5 := _t6 OR (_t5 AND K13);
_t36 := (_t6 OR (_t5 AND K13)) AND S4_2;
K6 := t6AfterTON.Q;
TO_LIST13 := _t141;
RV4TON(IN := _t36, PT := T#6s);
RV4 := RV4TON.Q;
KM11_1 := _t36;
_t46 := (NOT P0 AND _vacumContactOnDI AND NOT TRM7) AND NOT K13;
K7 := _t46 AND NOT RV5;
_t141 := _t36 AND K13;
t6AfterTON(IN := _t36, PT := T#5s);
K8 := (_t46 AND NOT RV5) AND S6_1;
RV5TON(IN := _t46, PT := T#90s);
RV5 := RV5TON.Q;
END_PROGRAM

(* POU L08, CFC *)
PROGRAM L08
VAR


END_VAR
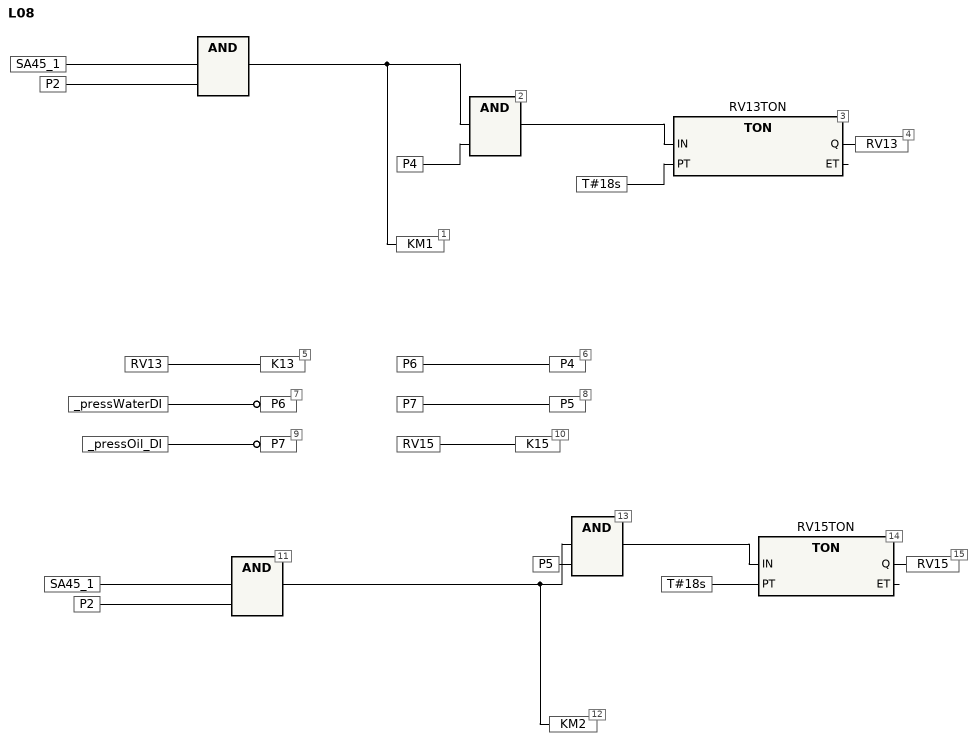
_CFC_ (* Continuous Function Chart, elements in execution order *)
#0 AND(SA45_1, P2)
#1 KM1 <= #0
#2 AND(#0, P4)
#3 RV13TON:TON(IN: #2, PT: T#18s)
#4 RV13 <= #3.Q
#5 K13 <= RV13
#6 P4 <= P6
#7 P6 <= NOT _pressWaterDI
#8 P5 <= P7
#9 P7 <= NOT _pressOil_DI
#10 K15 <= RV15
#11 AND(SA45_1, P2)
#12 KM2 <= #11
#13 AND(#11, P5)
#14 RV15TON:TON(IN: #13, PT: T#18s)
#15 RV15 <= #14.Q
_END_CFC_
(* the same logic as Structured Text *)
KM1 := SA45_1 AND P2;
RV13TON(IN := (SA45_1 AND P2) AND P4, PT := T#18s);
RV13 := RV13TON.Q;
K13 := RV13;
P4 := P6;
P6 := NOT _pressWaterDI;
P5 := P7;
P7 := NOT _pressOil_DI;
K15 := RV15;
KM2 := SA45_1 AND P2;
RV15TON(IN := (SA45_1 AND P2) AND P5, PT := T#18s);
RV15 := RV15TON.Q;
END_PROGRAM

(* POU L09, CFC *)
PROGRAM L09
VAR




	S18_1_prymoy: BOOL := TRUE;
END_VAR
VAR (* helpers for the ST form of the networks *)
	_t49 : BOOL;
END_VAR
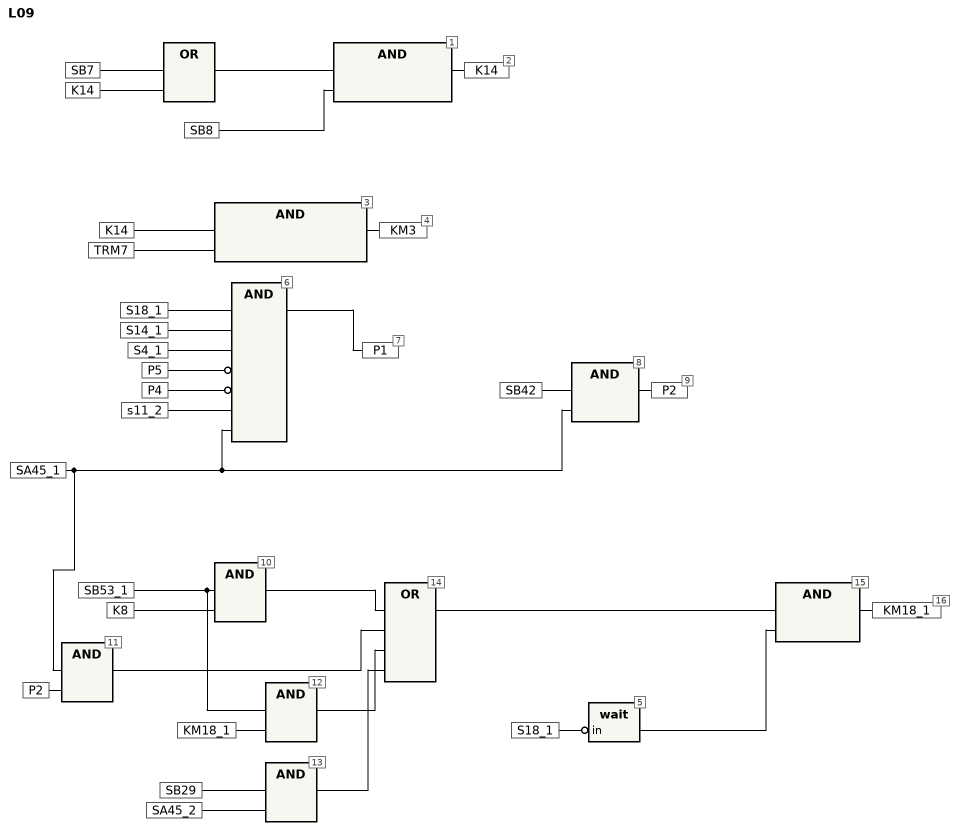
_CFC_ (* Continuous Function Chart, elements in execution order *)
#0 OR(SB7, K14)
#1 AND(#0, SB8)
#2 K14 <= #1
#3 AND(K14, TRM7)
#4 KM3 <= #3
#5 wait(in: NOT S18_1)
#6 AND(S18_1, S14_1, S4_1, NOT P5, NOT P4, s11_2, SA45_1)
#7 P1 <= #6
#8 AND(SB42, SA45_1)
#9 P2 <= #8
#10 AND(SB53_1, K8)
#11 AND(SA45_1, P2)
#12 AND(SB53_1, KM18_1)
#13 AND(SB29, SA45_2)
#14 OR(#10, #11, #12, #13)
#15 AND(#14, #5)
#16 KM18_1 <= #15
_END_CFC_
(* the same logic as Structured Text *)
K14 := (SB7 OR K14) AND SB8;
KM3 := K14 AND TRM7;
_t49 := wait(in := NOT S18_1);
P1 := S18_1 AND S14_1 AND S4_1 AND NOT P5 AND NOT P4 AND s11_2 AND SA45_1;
P2 := SB42 AND SA45_1;
KM18_1 := ((SB53_1 AND K8) OR (SA45_1 AND P2) OR (SB53_1 AND KM18_1) OR (SB29 AND SA45_2)) AND _t49;
END_PROGRAM

(* POU wait, LD *)
FUNCTION wait : BOOL
VAR_INPUT
	in : BOOL;
END_VAR
VAR
	vaqt : TIME := T#120s;
	tp1: TOF;
END_VAR
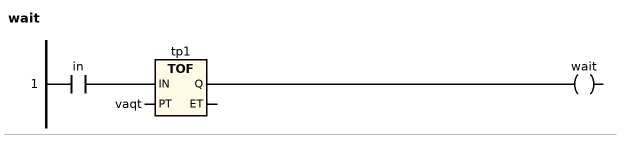
_LD_ (* Ladder Diagram *)
NETWORK 1
	[in] - tp1:TOF(IN: *, PT: vaqt) --- (wait)
_END_LD_
(* the same logic as Structured Text *)
(* Network 1 *)
tp1(IN := in, PT := vaqt);
wait := tp1.Q;
END_FUNCTION

(* POU L10, CFC *)
PROGRAM L10
VAR
	_17S_2: BOOL;

END_VAR
VAR (* helpers for the ST form of the networks *)
	_t68 : BOOL;
	_t69 : BOOL;
END_VAR
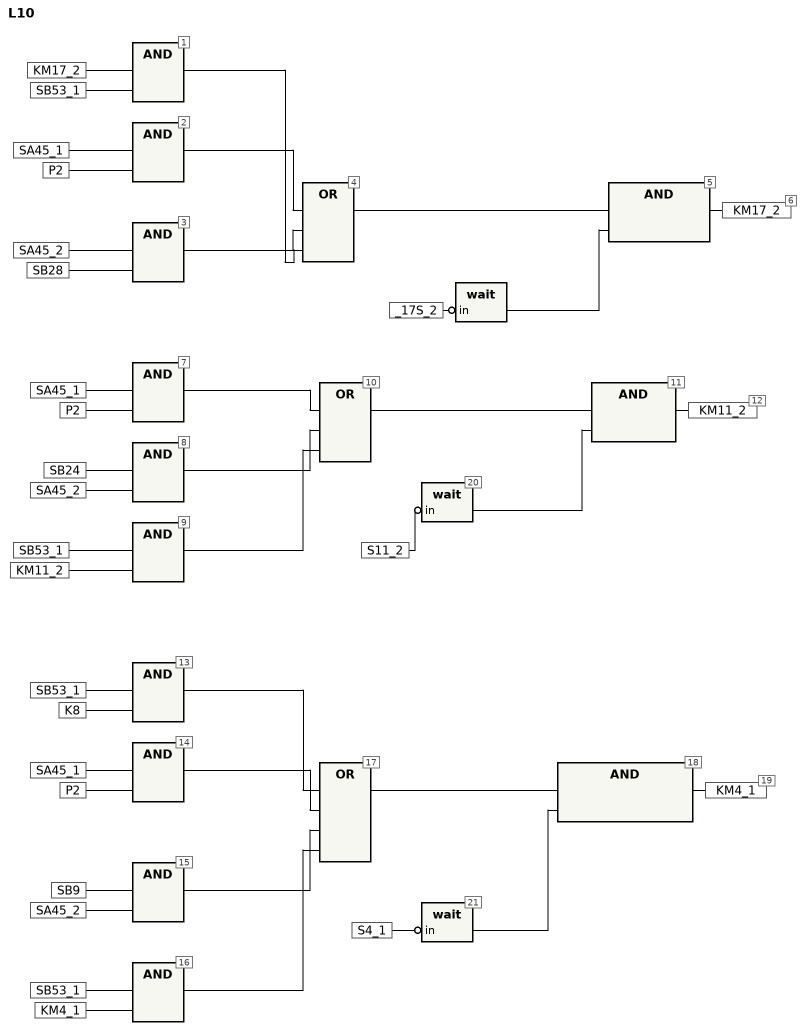
_CFC_ (* Continuous Function Chart, elements in execution order *)
#0 wait(in: NOT _17S_2)
#1 AND(KM17_2, SB53_1)
#2 AND(SA45_1, P2)
#3 AND(SA45_2, SB28)
#4 OR(#2, #3, #1)
#5 AND(#4, #0)
#6 KM17_2 <= #5
#7 AND(SA45_1, P2)
#8 AND(SB24, SA45_2)
#9 AND(SB53_1, KM11_2)
#10 OR(#7, #8, #9)
#11 AND(#10, #20)
#12 KM11_2 <= #11
#13 AND(SB53_1, K8)
#14 AND(SA45_1, P2)
#15 AND(SB9, SA45_2)
#16 AND(SB53_1, KM4_1)
#17 OR(#13, #14, #15, #16)
#18 AND(#17, #21)
#19 KM4_1 <= #18
#20 wait(in: NOT S11_2)
#21 wait(in: NOT S4_1)
_END_CFC_
(* the same logic as Structured Text *)
KM17_2 := ((SA45_1 AND P2) OR (SA45_2 AND SB28) OR (KM17_2 AND SB53_1)) AND wait(in := NOT _17S_2);
KM11_2 := ((SA45_1 AND P2) OR (SB24 AND SA45_2) OR (SB53_1 AND KM11_2)) AND _t68;
KM4_1 := ((SB53_1 AND K8) OR (SA45_1 AND P2) OR (SB9 AND SA45_2) OR (SB53_1 AND KM4_1)) AND _t69;
_t68 := wait(in := NOT S11_2);
_t69 := wait(in := NOT S4_1);
END_PROGRAM

(* POU L11, CFC *)
PROGRAM L11
VAR


	_16S_2: BOOL;
END_VAR
VAR (* helpers for the ST form of the networks *)
	_t55 : BOOL;
	_t54 : BOOL;
	_t36 : BOOL;
END_VAR
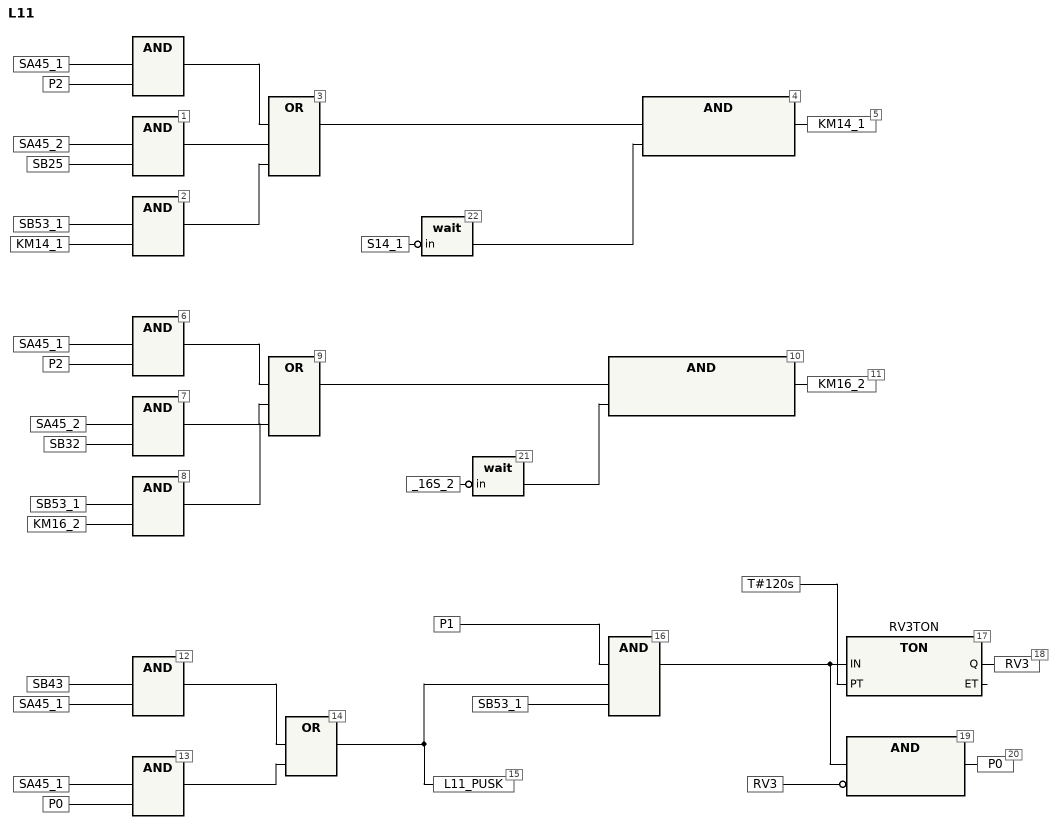
_CFC_ (* Continuous Function Chart, elements in execution order *)
#0 AND(SA45_1, P2)
#1 AND(SA45_2, SB25)
#2 AND(SB53_1, KM14_1)
#3 OR(#0, #1, #2)
#4 AND(#3, #22)
#5 KM14_1 <= #4
#6 AND(SA45_1, P2)
#7 AND(SA45_2, SB32)
#8 AND(SB53_1, KM16_2)
#9 OR(#6, #7, #8)
#10 AND(#9, #21)
#11 KM16_2 <= #10
#12 AND(SB43, SA45_1)
#13 AND(SA45_1, P0)
#14 OR(#12, #13)
#15 L11_PUSK <= #14
#16 AND(P1, #14, SB53_1)
#17 RV3TON:TON(IN: #16, PT: T#120s)
#18 RV3 <= #17.Q
#19 AND(#16, NOT RV3)
#20 P0 <= #19
#21 wait(in: NOT _16S_2)
#22 wait(in: NOT S14_1)
_END_CFC_
(* the same logic as Structured Text *)
KM14_1 := ((SA45_1 AND P2) OR (SA45_2 AND SB25) OR (SB53_1 AND KM14_1)) AND _t55;
KM16_2 := ((SA45_1 AND P2) OR (SA45_2 AND SB32) OR (SB53_1 AND KM16_2)) AND _t54;
_t36 := (SB43 AND SA45_1) OR (SA45_1 AND P0);
L11_PUSK := _t36;
RV3TON(IN := P1 AND _t36 AND SB53_1, PT := T#120s);
RV3 := RV3TON.Q;
P0 := (P1 AND _t36 AND SB53_1) AND NOT RV3;
_t54 := wait(in := NOT _16S_2);
_t55 := wait(in := NOT S14_1);
END_PROGRAM

(* POU L12, CFC *)
PROGRAM L12
VAR







END_VAR
VAR (* helpers for the ST form of the networks *)
	_t5 : BOOL;
	_t85 : BOOL;
	_t25 : BOOL;
	_t86 : BOOL;
	_t45 : BOOL;
	_t87 : BOOL;
	_t59 : BOOL;
	_t88 : BOOL;
END_VAR
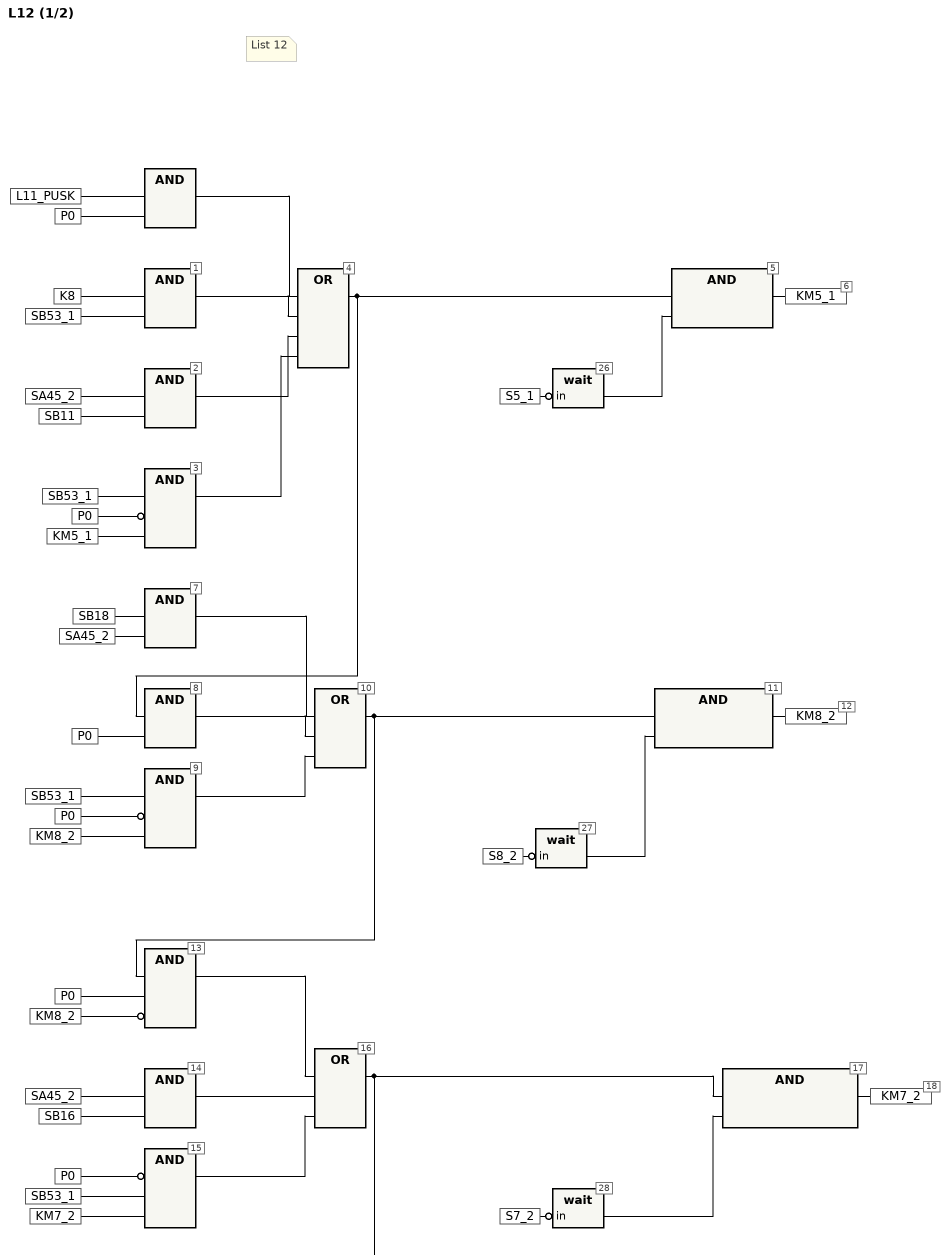
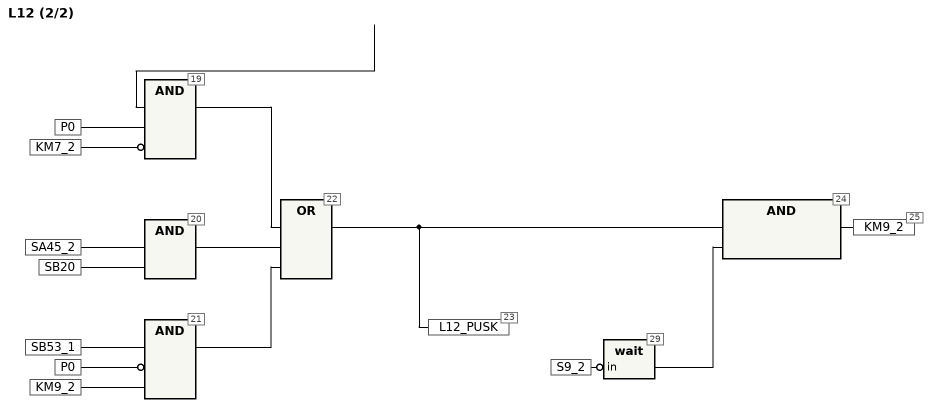
_CFC_ (* Continuous Function Chart, elements in execution order *)
(* List 12 *)
#0 AND(L11_PUSK, P0)
#1 AND(K8, SB53_1)
#2 AND(SA45_2, SB11)
#3 AND(SB53_1, NOT P0, KM5_1)
#4 OR(#0, #1, #2, #3)
#5 AND(#4, #26)
#6 KM5_1 <= #5
#7 AND(SB18, SA45_2)
#8 AND(#4, P0)
#9 AND(SB53_1, NOT P0, KM8_2)
#10 OR(#7, #8, #9)
#11 AND(#10, #27)
#12 KM8_2 <= #11
#13 AND(#10, P0, NOT KM8_2)
#14 AND(SA45_2, SB16)
#15 AND(NOT P0, SB53_1, KM7_2)
#16 OR(#13, #14, #15)
#17 AND(#16, #28)
#18 KM7_2 <= #17
#19 AND(#16, P0, NOT KM7_2)
#20 AND(SA45_2, SB20)
#21 AND(SB53_1, NOT P0, KM9_2)
#22 OR(#19, #20, #21)
#23 L12_PUSK <= #22
#24 AND(#22, #29)
#25 KM9_2 <= #24
#26 wait(in: NOT S5_1)
#27 wait(in: NOT S8_2)
#28 wait(in: NOT S7_2)
#29 wait(in: NOT S9_2)
_END_CFC_
(* the same logic as Structured Text *)
(* List 12 *)
_t5 := (L11_PUSK AND P0) OR (K8 AND SB53_1) OR (SA45_2 AND SB11) OR (SB53_1 AND NOT P0 AND KM5_1);
KM5_1 := _t5 AND _t85;
_t25 := (SB18 AND SA45_2) OR (_t5 AND P0) OR (SB53_1 AND NOT P0 AND KM8_2);
KM8_2 := _t25 AND _t86;
_t45 := (_t25 AND P0 AND NOT KM8_2) OR (SA45_2 AND SB16) OR (NOT P0 AND SB53_1 AND KM7_2);
KM7_2 := _t45 AND _t87;
_t59 := (_t45 AND P0 AND NOT KM7_2) OR (SA45_2 AND SB20) OR (SB53_1 AND NOT P0 AND KM9_2);
L12_PUSK := _t59;
KM9_2 := _t59 AND _t88;
_t85 := wait(in := NOT S5_1);
_t86 := wait(in := NOT S8_2);
_t87 := wait(in := NOT S7_2);
_t88 := wait(in := NOT S9_2);
END_PROGRAM

(* POU L13, CFC *)
PROGRAM L13
VAR



	P4: BOOL;

END_VAR
VAR (* helpers for the ST form of the networks *)
	_t12 : BOOL;
	_t20 : BOOL;
	_t19 : BOOL;
	_t23 : BOOL;
END_VAR
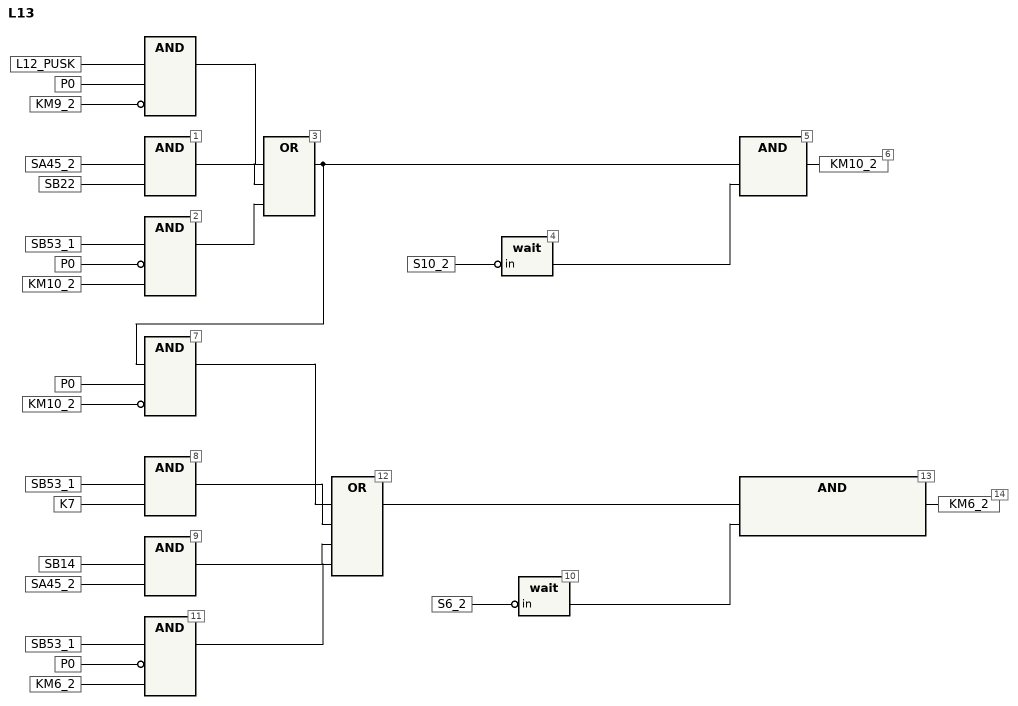
_CFC_ (* Continuous Function Chart, elements in execution order *)
#0 AND(L12_PUSK, P0, NOT KM9_2)
#1 AND(SA45_2, SB22)
#2 AND(SB53_1, NOT P0, KM10_2)
#3 OR(#0, #1, #2)
#4 wait(in: NOT S10_2)
#5 AND(#3, #4)
#6 KM10_2 <= #5
#7 AND(#3, P0, NOT KM10_2)
#8 AND(SB53_1, K7)
#9 AND(SB14, SA45_2)
#10 wait(in: NOT S6_2)
#11 AND(SB53_1, NOT P0, KM6_2)
#12 OR(#7, #8, #9, #11)
#13 AND(#12, #10)
#14 KM6_2 <= #13
_END_CFC_
(* the same logic as Structured Text *)
_t12 := (L12_PUSK AND P0 AND NOT KM9_2) OR (SA45_2 AND SB22) OR (SB53_1 AND NOT P0 AND KM10_2);
KM10_2 := _t12 AND wait(in := NOT S10_2);
_t20 := _t12 AND P0 AND NOT KM10_2;
_t19 := SB53_1 AND K7;
_t23 := SB14 AND SA45_2;
KM6_2 := (_t20 OR _t19 OR _t23 OR (SB53_1 AND NOT P0 AND KM6_2)) AND wait(in := NOT S6_2);
END_PROGRAM

(* POU L14, CFC *)
PROGRAM L14
VAR

END_VAR
VAR (* helpers for the ST form of the networks *)
	_t6 : BOOL;
	_t29 : BOOL;
END_VAR
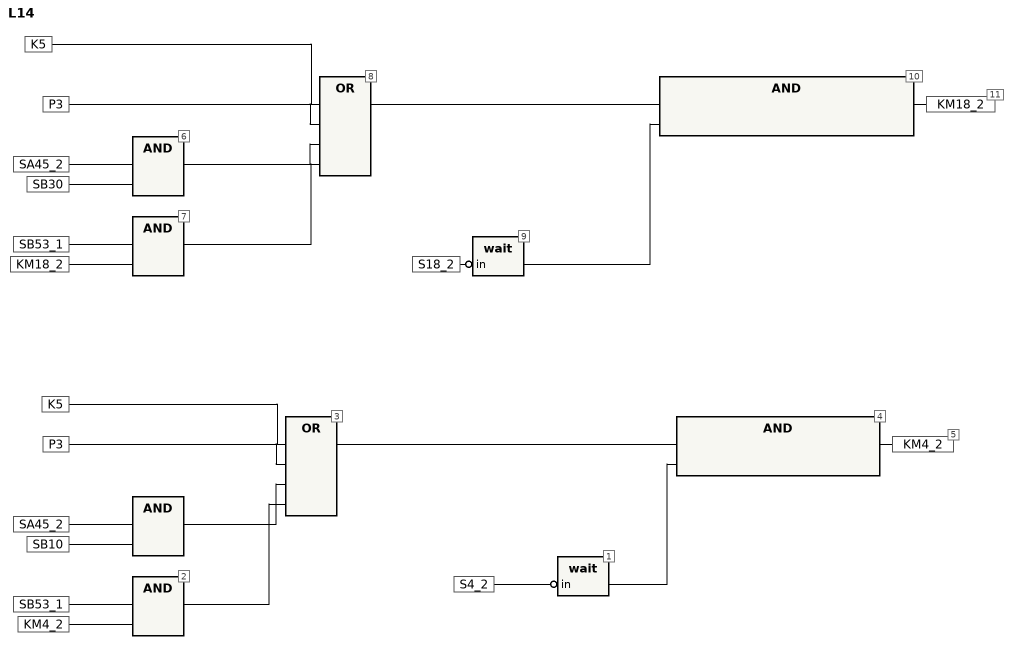
_CFC_ (* Continuous Function Chart, elements in execution order *)
#0 AND(SA45_2, SB10)
#1 wait(in: NOT S4_2)
#2 AND(SB53_1, KM4_2)
#3 OR(K5, P3, #0, #2)
#4 AND(#3, #1)
#5 KM4_2 <= #4
#6 AND(SA45_2, SB30)
#7 AND(SB53_1, KM18_2)
#8 OR(K5, P3, #6, #7)
#9 wait(in: NOT S18_2)
#10 AND(#8, #9)
#11 KM18_2 <= #10
_END_CFC_
(* the same logic as Structured Text *)
_t6 := SA45_2 AND SB10;
KM4_2 := (K5 OR P3 OR _t6 OR (SB53_1 AND KM4_2)) AND wait(in := NOT S4_2);
_t29 := K5 OR P3 OR (SA45_2 AND SB30) OR (SB53_1 AND KM18_2);
KM18_2 := _t29 AND wait(in := NOT S18_2);
END_PROGRAM

(* POU L15, CFC *)
PROGRAM L15
VAR

END_VAR
VAR (* helpers for the ST form of the networks *)
	_t14 : BOOL;
	_t20 : BOOL;
	_t28 : BOOL;
	_t34 : BOOL;
	_t46 : BOOL;
END_VAR
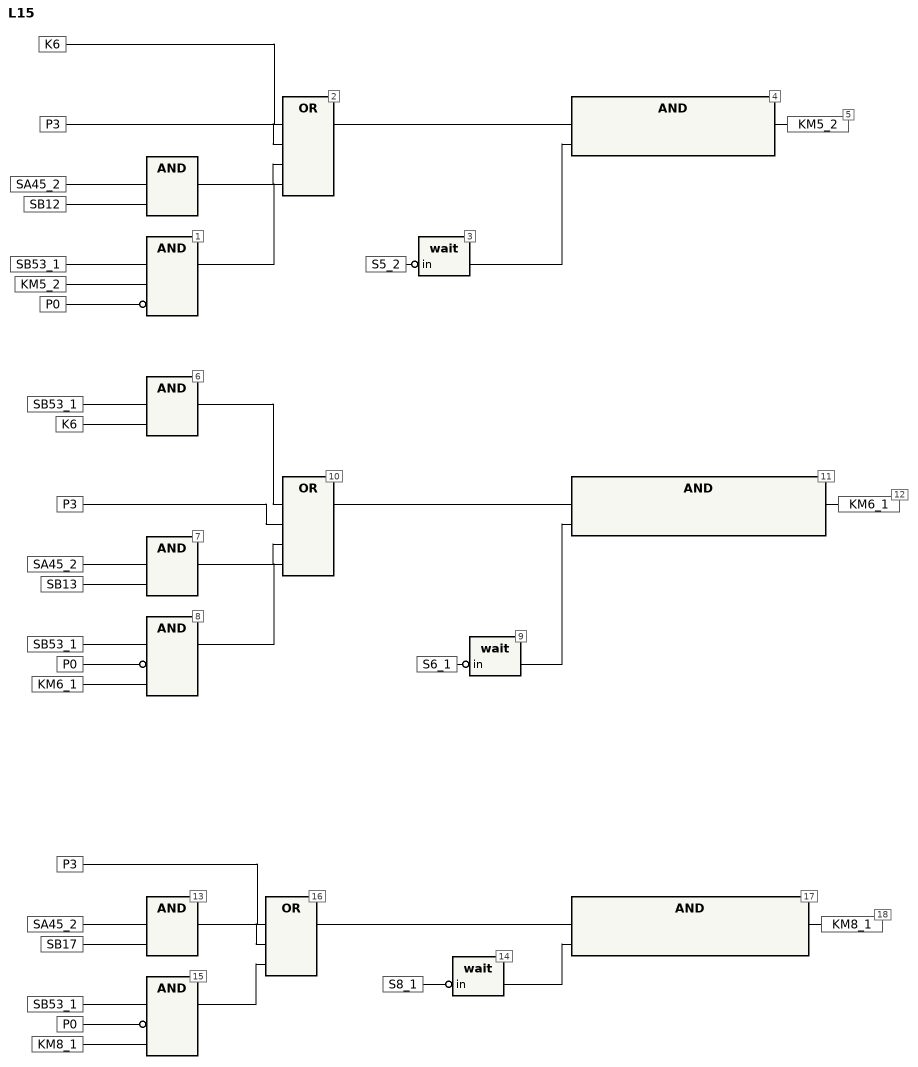
_CFC_ (* Continuous Function Chart, elements in execution order *)
#0 AND(SA45_2, SB12)
#1 AND(SB53_1, KM5_2, NOT P0)
#2 OR(K6, P3, #0, #1)
#3 wait(in: NOT S5_2)
#4 AND(#2, #3)
#5 KM5_2 <= #4
#6 AND(SB53_1, K6)
#7 AND(SA45_2, SB13)
#8 AND(SB53_1, NOT P0, KM6_1)
#9 wait(in: NOT S6_1)
#10 OR(#6, P3, #7, #8)
#11 AND(#10, #9)
#12 KM6_1 <= #11
#13 AND(SA45_2, SB17)
#14 wait(in: NOT S8_1)
#15 AND(SB53_1, NOT P0, KM8_1)
#16 OR(P3, #13, #15)
#17 AND(#16, #14)
#18 KM8_1 <= #17
_END_CFC_
(* the same logic as Structured Text *)
_t14 := K6 OR P3 OR (SA45_2 AND SB12) OR (SB53_1 AND KM5_2 AND NOT P0);
KM5_2 := _t14 AND wait(in := NOT S5_2);
_t20 := SB53_1 AND K6;
_t28 := SA45_2 AND SB13;
_t34 := SB53_1 AND NOT P0 AND KM6_1;
KM6_1 := (_t20 OR P3 OR _t28 OR _t34) AND wait(in := NOT S6_1);
_t46 := SA45_2 AND SB17;
KM8_1 := (P3 OR _t46 OR (SB53_1 AND NOT P0 AND KM8_1)) AND wait(in := NOT S8_1);
END_PROGRAM

(* POU L16, CFC *)
PROGRAM L16
VAR
	mt7TON: TON;

	mt9TON: TON;
	mt10TON: TON;
END_VAR
VAR (* helpers for the ST form of the networks *)
	_t3 : BOOL;
	_t51 : BOOL;
	_t81 : BOOL;
	_t96 : BOOL;
	_t126 : BOOL;
END_VAR
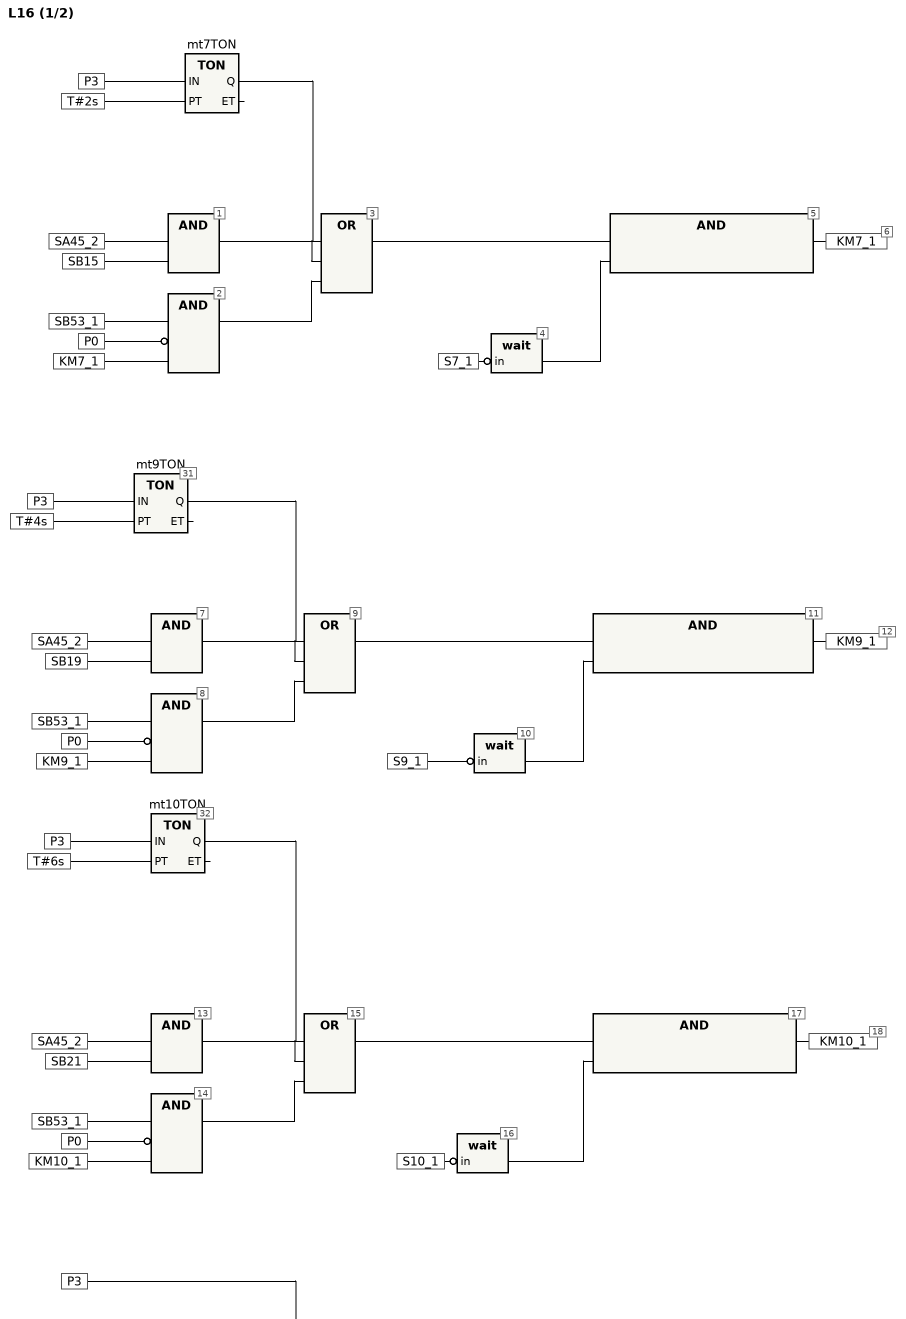
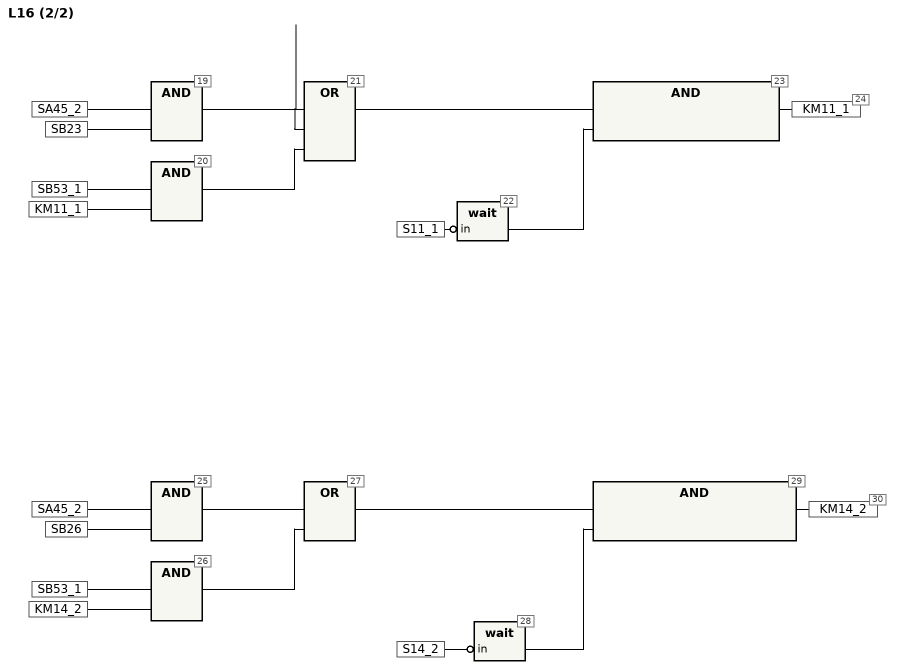
_CFC_ (* Continuous Function Chart, elements in execution order *)
#0 mt7TON:TON(IN: P3, PT: T#2s)
#1 AND(SA45_2, SB15)
#2 AND(SB53_1, NOT P0, KM7_1)
#3 OR(#0.Q, #1, #2)
#4 wait(in: NOT S7_1)
#5 AND(#3, #4)
#6 KM7_1 <= #5
#7 AND(SA45_2, SB19)
#8 AND(SB53_1, NOT P0, KM9_1)
#9 OR(#31.Q, #7, #8)
#10 wait(in: NOT S9_1)
#11 AND(#9, #10)
#12 KM9_1 <= #11
#13 AND(SA45_2, SB21)
#14 AND(SB53_1, NOT P0, KM10_1)
#15 OR(#32.Q, #13, #14)
#16 wait(in: NOT S10_1)
#17 AND(#15, #16)
#18 KM10_1 <= #17
#19 AND(SA45_2, SB23)
#20 AND(SB53_1, KM11_1)
#21 OR(P3, #19, #20)
#22 wait(in: NOT S11_1)
#23 AND(#21, #22)
#24 KM11_1 <= #23
#25 AND(SA45_2, SB26)
#26 AND(SB53_1, KM14_2)
#27 OR(#25, #26)
#28 wait(in: NOT S14_2)
#29 AND(#27, #28)
#30 KM14_2 <= #29
#31 mt9TON:TON(IN: P3, PT: T#4s)
#32 mt10TON:TON(IN: P3, PT: T#6s)
_END_CFC_
(* the same logic as Structured Text *)
mt7TON(IN := P3, PT := T#2s);
_t3 := mt7TON.Q OR (SA45_2 AND SB15) OR (SB53_1 AND NOT P0 AND KM7_1);
KM7_1 := _t3 AND wait(in := NOT S7_1);
_t51 := mt9TON.Q OR (SA45_2 AND SB19) OR (SB53_1 AND NOT P0 AND KM9_1);
KM9_1 := _t51 AND wait(in := NOT S9_1);
_t81 := mt10TON.Q OR (SA45_2 AND SB21) OR (SB53_1 AND NOT P0 AND KM10_1);
KM10_1 := _t81 AND wait(in := NOT S10_1);
_t96 := P3 OR (SA45_2 AND SB23) OR (SB53_1 AND KM11_1);
KM11_1 := _t96 AND wait(in := NOT S11_1);
_t126 := (SA45_2 AND SB26) OR (SB53_1 AND KM14_2);
KM14_2 := _t126 AND wait(in := NOT S14_2);
mt9TON(IN := P3, PT := T#4s);
mt10TON(IN := P3, PT := T#6s);
END_PROGRAM

(* POU gatesAlarm, LD *)
PROGRAM gatesAlarm
VAR
	al1: alarm;
	al18_2: alarm;
	al18_1: alarm;
	al4_1: alarm;
	al4_2: alarm;
	al5_1: alarm;
	al5_2: alarm;
	al6_1: alarm;
	al6_2: alarm;
	al7_2: alarm;
	al7_1: alarm;
	al8_1: alarm;
	al8_2: alarm;
	al9_1: alarm;
	al9_2: alarm;
	al10_1: alarm;
	al10_2: alarm;
	a11_1: alarm;
	al11_2: alarm;
	al14_1: alarm;
	al14_2: alarm;
	vaqt : WORD := 70;
END_VAR
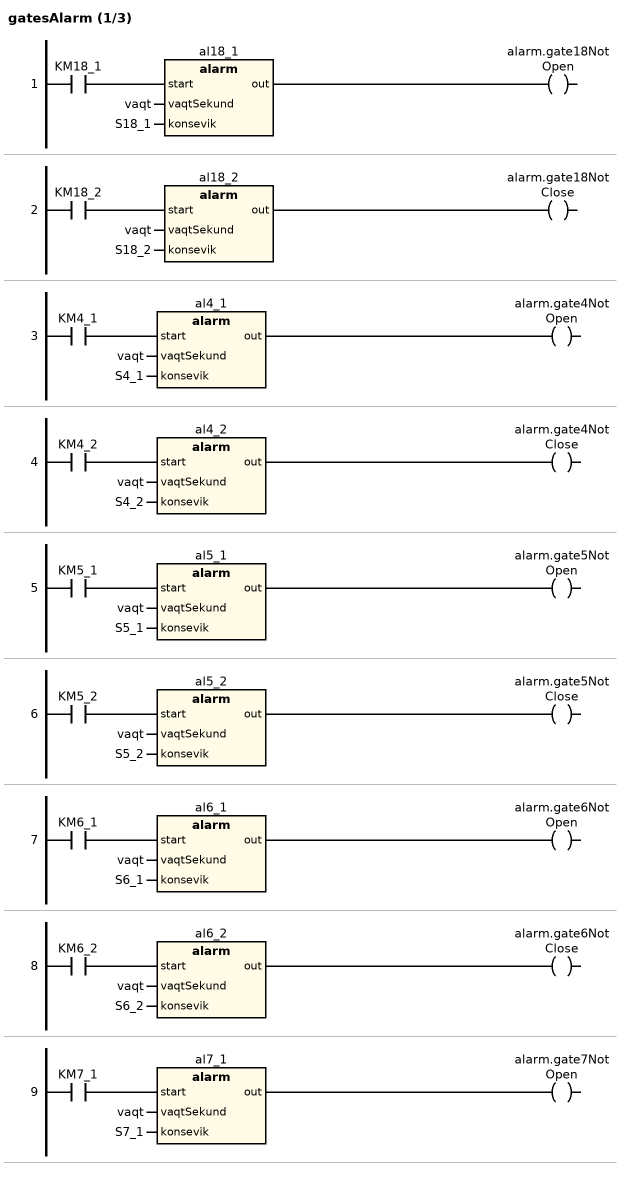
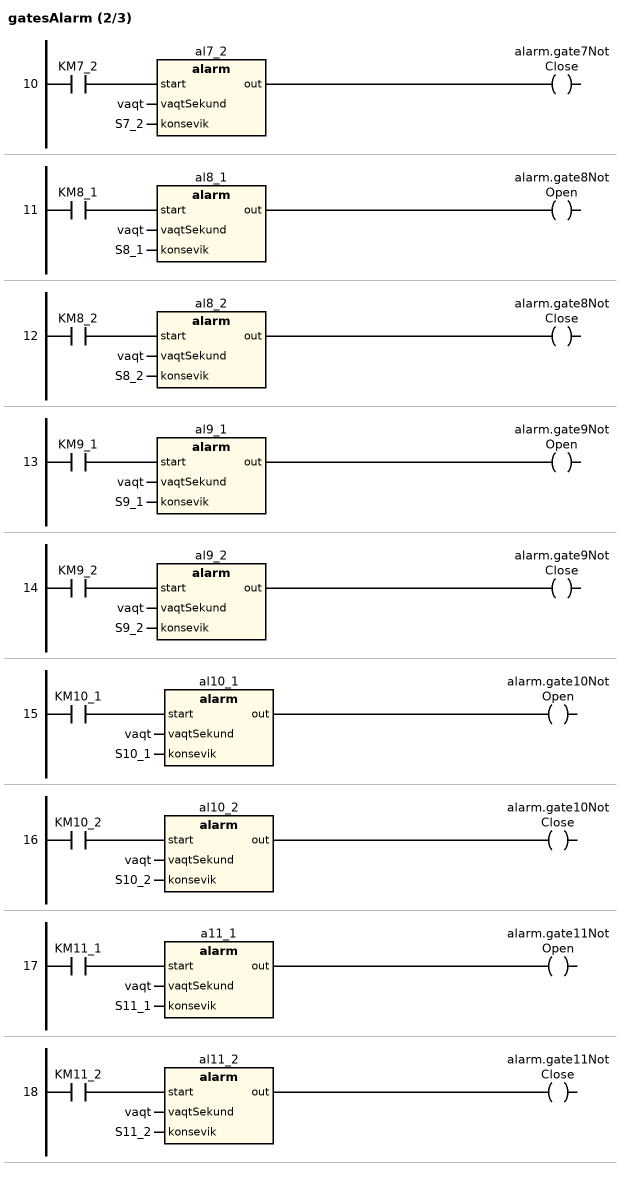
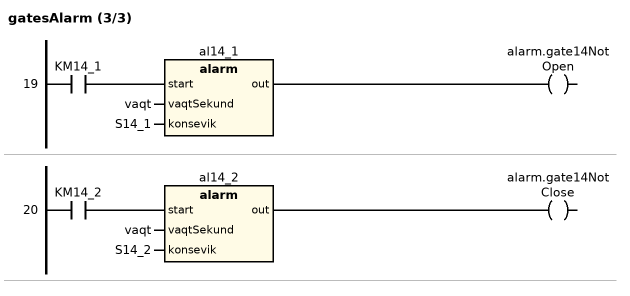
_LD_ (* Ladder Diagram *)
NETWORK 1
	[KM18_1] - al18_1:alarm(start: *, vaqtSekund: vaqt, konsevik: S18_1) --- (alarm.gate18NotOpen)
NETWORK 2
	[KM18_2] - al18_2:alarm(start: *, vaqtSekund: vaqt, konsevik: S18_2) --- (alarm.gate18NotClose)
NETWORK 3
	[KM4_1] - al4_1:alarm(start: *, vaqtSekund: vaqt, konsevik: S4_1) --- (alarm.gate4NotOpen)
NETWORK 4
	[KM4_2] - al4_2:alarm(start: *, vaqtSekund: vaqt, konsevik: S4_2) --- (alarm.gate4NotClose)
NETWORK 5
	[KM5_1] - al5_1:alarm(start: *, vaqtSekund: vaqt, konsevik: S5_1) --- (alarm.gate5NotOpen)
NETWORK 6
	[KM5_2] - al5_2:alarm(start: *, vaqtSekund: vaqt, konsevik: S5_2) --- (alarm.gate5NotClose)
NETWORK 7
	[KM6_1] - al6_1:alarm(start: *, vaqtSekund: vaqt, konsevik: S6_1) --- (alarm.gate6NotOpen)
NETWORK 8
	[KM6_2] - al6_2:alarm(start: *, vaqtSekund: vaqt, konsevik: S6_2) --- (alarm.gate6NotClose)
NETWORK 9
	[KM7_1] - al7_1:alarm(start: *, vaqtSekund: vaqt, konsevik: S7_1) --- (alarm.gate7NotOpen)
NETWORK 10
	[KM7_2] - al7_2:alarm(start: *, vaqtSekund: vaqt, konsevik: S7_2) --- (alarm.gate7NotClose)
NETWORK 11
	[KM8_1] - al8_1:alarm(start: *, vaqtSekund: vaqt, konsevik: S8_1) --- (alarm.gate8NotOpen)
NETWORK 12
	[KM8_2] - al8_2:alarm(start: *, vaqtSekund: vaqt, konsevik: S8_2) --- (alarm.gate8NotClose)
NETWORK 13
	[KM9_1] - al9_1:alarm(start: *, vaqtSekund: vaqt, konsevik: S9_1) --- (alarm.gate9NotOpen)
NETWORK 14
	[KM9_2] - al9_2:alarm(start: *, vaqtSekund: vaqt, konsevik: S9_2) --- (alarm.gate9NotClose)
NETWORK 15
	[KM10_1] - al10_1:alarm(start: *, vaqtSekund: vaqt, konsevik: S10_1) --- (alarm.gate10NotOpen)
NETWORK 16
	[KM10_2] - al10_2:alarm(start: *, vaqtSekund: vaqt, konsevik: S10_2) --- (alarm.gate10NotClose)
NETWORK 17
	[KM11_1] - a11_1:alarm(start: *, vaqtSekund: vaqt, konsevik: S11_1) --- (alarm.gate11NotOpen)
NETWORK 18
	[KM11_2] - al11_2:alarm(start: *, vaqtSekund: vaqt, konsevik: S11_2) --- (alarm.gate11NotClose)
NETWORK 19
	[KM14_1] - al14_1:alarm(start: *, vaqtSekund: vaqt, konsevik: S14_1) --- (alarm.gate14NotOpen)
NETWORK 20
	[KM14_2] - al14_2:alarm(start: *, vaqtSekund: vaqt, konsevik: S14_2) --- (alarm.gate14NotClose)
_END_LD_
(* the same logic as Structured Text *)
(* Network 1 *)
al18_1(start := KM18_1, vaqtSekund := vaqt, konsevik := S18_1);
alarm.gate18NotOpen := al18_1.out;
(* Network 2 *)
al18_2(start := KM18_2, vaqtSekund := vaqt, konsevik := S18_2);
alarm.gate18NotClose := al18_2.out;
(* Network 3 *)
al4_1(start := KM4_1, vaqtSekund := vaqt, konsevik := S4_1);
alarm.gate4NotOpen := al4_1.out;
(* Network 4 *)
al4_2(start := KM4_2, vaqtSekund := vaqt, konsevik := S4_2);
alarm.gate4NotClose := al4_2.out;
(* Network 5 *)
al5_1(start := KM5_1, vaqtSekund := vaqt, konsevik := S5_1);
alarm.gate5NotOpen := al5_1.out;
(* Network 6 *)
al5_2(start := KM5_2, vaqtSekund := vaqt, konsevik := S5_2);
alarm.gate5NotClose := al5_2.out;
(* Network 7 *)
al6_1(start := KM6_1, vaqtSekund := vaqt, konsevik := S6_1);
alarm.gate6NotOpen := al6_1.out;
(* Network 8 *)
al6_2(start := KM6_2, vaqtSekund := vaqt, konsevik := S6_2);
alarm.gate6NotClose := al6_2.out;
(* Network 9 *)
al7_1(start := KM7_1, vaqtSekund := vaqt, konsevik := S7_1);
alarm.gate7NotOpen := al7_1.out;
(* Network 10 *)
al7_2(start := KM7_2, vaqtSekund := vaqt, konsevik := S7_2);
alarm.gate7NotClose := al7_2.out;
(* Network 11 *)
al8_1(start := KM8_1, vaqtSekund := vaqt, konsevik := S8_1);
alarm.gate8NotOpen := al8_1.out;
(* Network 12 *)
al8_2(start := KM8_2, vaqtSekund := vaqt, konsevik := S8_2);
alarm.gate8NotClose := al8_2.out;
(* Network 13 *)
al9_1(start := KM9_1, vaqtSekund := vaqt, konsevik := S9_1);
alarm.gate9NotOpen := al9_1.out;
(* Network 14 *)
al9_2(start := KM9_2, vaqtSekund := vaqt, konsevik := S9_2);
alarm.gate9NotClose := al9_2.out;
(* Network 15 *)
al10_1(start := KM10_1, vaqtSekund := vaqt, konsevik := S10_1);
alarm.gate10NotOpen := al10_1.out;
(* Network 16 *)
al10_2(start := KM10_2, vaqtSekund := vaqt, konsevik := S10_2);
alarm.gate10NotClose := al10_2.out;
(* Network 17 *)
a11_1(start := KM11_1, vaqtSekund := vaqt, konsevik := S11_1);
alarm.gate11NotOpen := a11_1.out;
(* Network 18 *)
al11_2(start := KM11_2, vaqtSekund := vaqt, konsevik := S11_2);
alarm.gate11NotClose := al11_2.out;
(* Network 19 *)
al14_1(start := KM14_1, vaqtSekund := vaqt, konsevik := S14_1);
alarm.gate14NotOpen := al14_1.out;
(* Network 20 *)
al14_2(start := KM14_2, vaqtSekund := vaqt, konsevik := S14_2);
alarm.gate14NotClose := al14_2.out;
END_PROGRAM

(* POU start_or_stop, LD *)
PROGRAM start_or_stop
VAR
	_controlFazaDI46: BOOL;
	kompressorOFF: TP;
	kompressorON: TP;
	_currentHighJD5DI00000: BOOL;
	P300000: BOOL;
	P00000: BOOL;

	alarmLedDO_MB555: BOOL;
	_kompOffDO_55555555: BOOL;
	_kompOnDO_555555: BOOL;
	trig: R_TRIG;

END_VAR
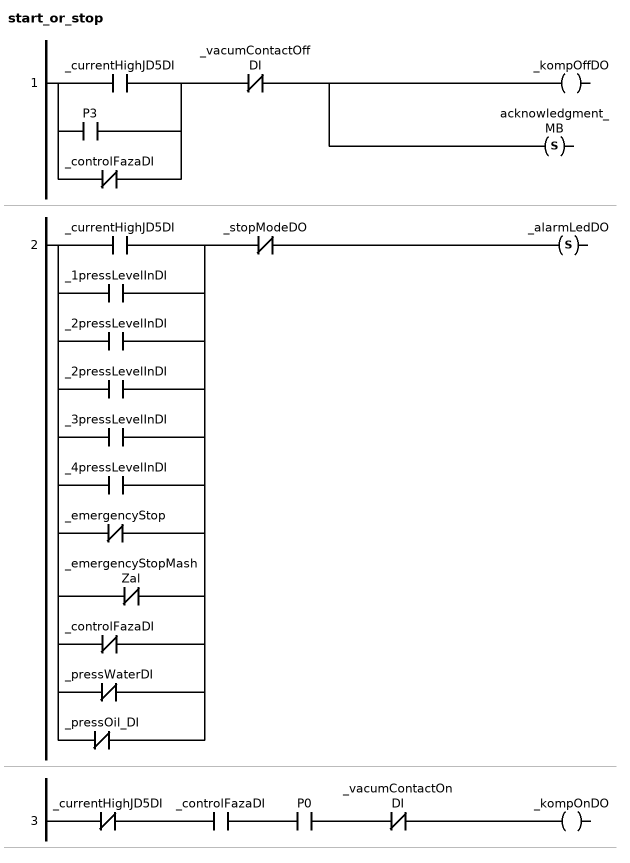
_LD_ (* Ladder Diagram *)
NETWORK 1
	{ [_currentHighJD5DI] | [P3] | [/_controlFazaDI] } - [/_vacumContactOffDI] --- (_kompOffDO) (S acknowledgment_MB)
NETWORK 2
	{ [_currentHighJD5DI] | [_1pressLevelInDI] | [_2pressLevelInDI] | [_2pressLevelInDI] | [_3pressLevelInDI] | [_4pressLevelInDI] | [/_emergencyStop] | [/_emergencyStopMashZal] | [/_controlFazaDI] | [/_pressWaterDI] | [/_pressOil_DI] } - [/_stopModeDO] --- (S _alarmLedDO)
NETWORK 3
	[/_currentHighJD5DI] - [_controlFazaDI] - [P0] - [/_vacumContactOnDI] --- (_kompOnDO)
_END_LD_
(* the same logic as Structured Text *)
(* Network 1 *)
_kompOffDO := (_currentHighJD5DI OR P3 OR NOT _controlFazaDI) AND NOT _vacumContactOffDI;
IF _kompOffDO THEN acknowledgment_MB := TRUE; END_IF;
(* Network 2 *)
IF (_currentHighJD5DI OR _1pressLevelInDI OR _2pressLevelInDI OR _2pressLevelInDI OR _3pressLevelInDI OR _4pressLevelInDI OR NOT _emergencyStop OR NOT _emergencyStopMashZal OR NOT _controlFazaDI OR NOT _pressWaterDI OR NOT _pressOil_DI) AND NOT _stopModeDO THEN _alarmLedDO := TRUE; END_IF;
(* Network 3 *)
_kompOnDO := NOT _currentHighJD5DI AND _controlFazaDI AND P0 AND NOT _vacumContactOnDI;
END_PROGRAM

(* POU E_STOP, LD *)
PROGRAM E_STOP
VAR
	P4: BOOL;
	tof1: TON;
	rtrig: R_TRIG;
	xato : ARRAY [0..17] OF BOOL;
	ton1 : TON;
END_VAR
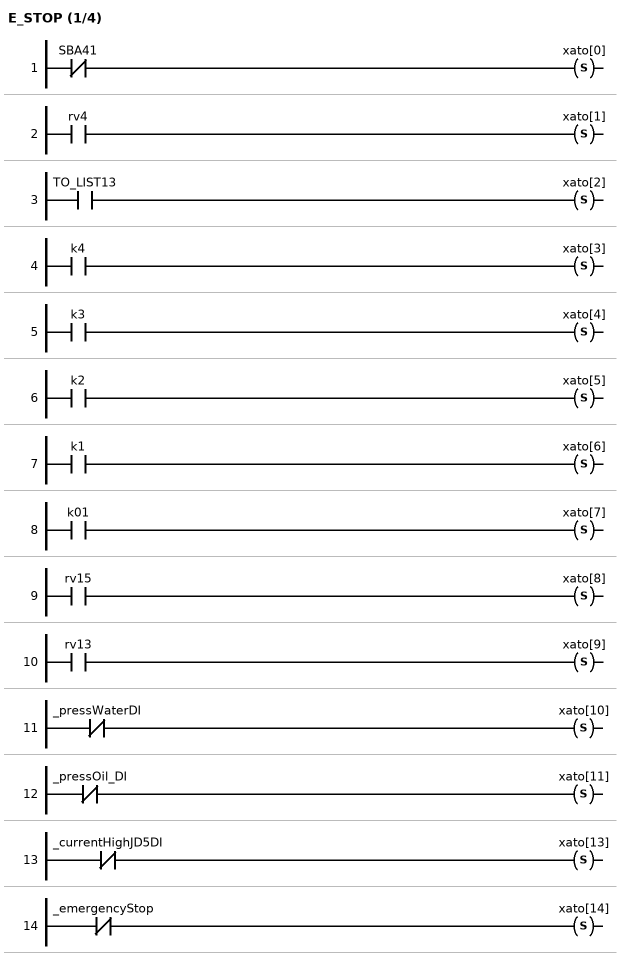
